LIN {X 0,Y 641.298,Z 835.183,A -85,B 0,C 180,E1 28744.796,E2 28744.796} C_VEL
LIN {X 0,Y 639.476,Z 856.383,A -85,B 0,C 180,E1 28743.716,E2 28743.716} C_VEL
LIN {X 0,Y 637.654,Z 876.672,A -85,B 0,C 180,E1 28742.537,E2 28742.537} C_VEL
LIN {X 0,Y 635.475,Z 900.138,A -85,B 0,C 180,E1 28740.959,E2 28740.959} C_VEL
LIN {X 0,Y 633.786,Z 917.988,A -85,B 0,C 180,E1 28739.591,E2 28739.591} C_VEL
LIN {X 0,Y 632.015,Z 936.849,A -85,B 0,C 180,E1 28737.975,E2 28737.975} C_VEL
LIN {X 0,Y 630.246,Z 955.886,A -85,B 0,C 180,E1 28736.108,E2 28736.108} C_VEL
LIN {X 0,Y 628.902,Z 971.248,A -85,B 0,C 180,E1 28734.417,E2 28734.417} C_VEL
LIN {X 0,Y 627.491,Z 988.385,A -85,B 0,C 180,E1 28732.287,E2 28732.287} C_VEL
LIN {X 0,Y 626.478,Z 1001.923,A -85,B 0,C 180,E1 28730.361,E2 28730.361} C_VEL
LIN {X 0,Y 625.634,Z 1015.034,A -85,B 0,C 180,E1 28728.255,E2 28728.255} C_VEL
LIN {X 0,Y 624.945,Z 1027.385,A -85,B 0,C 180,E1 28725.933,E2 28725.933} C_VEL
LIN {X 0,Y 624.537,Z 1036.289,A -85,B 0,C 180,E1 28723.99,E2 28723.99} C_VEL
LIN {X 0,Y 624.242,Z 1045.129,A -85,B 0,C 180,E1 28721.737,E2 28721.737} C_VEL
LIN {X 0,Y 624.044,Z 1052.386,A -85,B 0,C 180,E1 28719.406,E2 28719.406} C_VEL
LIN {X 0,Y 623.966,Z 1057.241,A -85,B 0,C 180,E1 28717.458,E2 28717.458} C_VEL
LIN {X 0,Y 623.913,Z 1061.124,A -85,B 0,C 180,E1 28715.426,E2 28715.426} C_VEL
LIN {X 0,Y 623.915,Z 1064.167,A -85,B 0,C 180,E1 28712.94,E2 28712.94} C_VEL
LIN {X 0,Y 623.908,Z 1065.282,A -85,B 0,C 180,E1 28710.918,E2 28710.918} C_VEL
LIN {X 0,Y 623.913,Z 1065.26,A -85,B 0,C 180,E1 28708.99,E2 28708.99} C_VEL
LIN {X 0,Y 623.908,Z 1063.894,A -85,B 0,C 180,E1 28706.693,E2 28706.693} C_VEL
LIN {X 0,Y 623.91,Z 1060.804,A -85,B 0,C 180,E1 28704.39,E2 28704.39} C_VEL
LIN {X 0,Y 623.968,Z 1057.034,A -85,B 0,C 180,E1 28702.449,E2 28702.449} C_VEL
LIN {X 0,Y 624.044,Z 1052.131,A -85,B 0,C 180,E1 28700.501,E2 28700.501} C_VEL
LIN {X 0,Y 624.249,Z 1044.691,A -85,B 0,C 180,E1 28698.146,E2 28698.146} C_VEL
LIN {X 0,Y 624.542,Z 1036.159,A -85,B 0,C 180,E1 28695.98,E2 28695.98} C_VEL
LIN {X 0,Y 624.955,Z 1027.192,A -85,B 0,C 180,E1 28694.027,E2 28694.027} C_VEL
LIN {X 0,Y 625.655,Z 1014.638,A -85,B 0,C 180,E1 28691.678,E2 28691.678} C_VEL
LIN {X 0,Y 626.478,Z 1001.926,A -85,B 0,C 180,E1 28689.639,E2 28689.639} C_VEL
LIN {X 0,Y 627.49,Z 988.385,A -85,B 0,C 180,E1 28687.713,E2 28687.713} C_VEL
LIN {X 0,Y 628.903,Z 971.248,A -85,B 0,C 180,E1 28685.583,E2 28685.583} C_VEL
LIN {X 0,Y 630.247,Z 955.885,A -85,B 0,C 180,E1 28683.892,E2 28683.892} C_VEL
LIN {X 0,Y 632.014,Z 936.851,A -85,B 0,C 180,E1 28682.025,E2 28682.025} C_VEL
LIN {X 0,Y 633.784,Z 917.986,A -85,B 0,C 180,E1 28680.409,E2 28680.409} C_VEL
LIN {X 0,Y 635.482,Z 900.053,A -85,B 0,C 180,E1 28679.035,E2 28679.035} C_VEL
LIN {X 0,Y 637.655,Z 876.666,A -85,B 0,C 180,E1 28677.463,E2 28677.463} C_VEL
LIN {X 0,Y 639.476,Z 856.385,A -85,B 0,C 180,E1 28676.284,E2 28676.284} C_VEL
LIN {X 0,Y 641.298,Z 835.19,A -85,B 0,C 180,E1 28675.204,E2 28675.204} C_VEL
LIN {X 0,Y 643.222,Z 810.081,A -85,B 0,C 180,E1 28674.123,E2 28674.123} C_VEL
LIN {X 0,Y 644.618,Z 789.698,A -85,B 0,C 180,E1 28673.387,E2 28673.387} C_VEL
LIN {X 0,Y 645.855,Z 769.341,A -85,B 0,C 180,E1 28672.768,E2 28672.768} C_VEL
LIN {X 0,Y 647.121,Z 744.666,A -85,B 0,C 180,E1 28672.163,E2 28672.163} C_VEL
LIN {X 0,Y 648.017,Z 719.173,A -85,B 0,C 180,E1 28671.716,E2 28671.716} C_VEL
LIN {X 0,Y 651.905,Z 492.19,A -85,B 0,C 180,E1 28668.782,E2 28668.782} C_VEL
LIN {X 0,Y 654.852,Z 321.153,A -85,B 0,C 180,E1 28666.527,E2 28666.527} C_VEL
LIN {X 0,Y 651.999,Z 316.125,A -85,B 0,C 180,E1 28666.214,E2 28666.214} C_VEL
LIN {X 0,Y 636.119,Z 291.599,A -85,B 0,C 180,E1 28664.466,E2 28664.466} C_VEL
LIN {X 0,Y 633.043,Z 286.91,A -85,B 0,C 180,E1 28664.089,E2 28664.089} C_VEL
LIN {X 0,Y 626.285,Z 271.766,A -85,B 0,C 180,E1 28662.11,E2 28662.11} C_VEL
LIN {X 0,Y 624.92,Z 268.282,A -85,B 0,C 180,E1 28661.607,E2 28661.607} C_VEL
LIN {X 0,Y 624.891,Z 268.104,A -85,B 0,C 180,E1 28658.368,E2 28658.368} C_VEL
LIN {X 0,Y 624.891,Z 268.132,A -85,B 0,C 180,E1 28655.622,E2 28655.622} C_VEL
LIN {X 0,Y 624.899,Z 268.127,A -85,B 0,C 180,E1 28652.346,E2 28652.346} C_VEL
LIN {X 0,Y 624.882,Z 268.114,A -85,B 0,C 180,E1 28649.633,E2 28649.633} C_VEL
LIN {X 0,Y 624.93,Z 268.128,A -85,B 0,C 180,E1 28646.513,E2 28646.513} C_VEL
LIN {X 0,Y 624.882,Z 268.129,A -85,B 0,C 180,E1 28643.58,E2 28643.58} C_VEL
LIN {X 0,Y 624.942,Z 268.125,A -85,B 0,C 180,E1 28640.512,E2 28640.512} C_VEL
LIN {X 0,Y 624.881,Z 268.136,A -85,B 0,C 180,E1 28637.603,E2 28637.603} C_VEL
LIN {X 0,Y 624.959,Z 268.135,A -85,B 0,C 180,E1 28634.545,E2 28634.545} C_VEL
LIN {X 0,Y 624.88,Z 268.136,A -85,B 0,C 180,E1 28631.538,E2 28631.538} C_VEL
LIN {X 0,Y 624.955,Z 268.121,A -85,B 0,C 180,E1 28628.464,E2 28628.464} C_VEL
LIN {X 0,Y 624.879,Z 268.136,A -85,B 0,C 180,E1 28625.509,E2 28625.509} C_VEL
LIN {X 0,Y 624.949,Z 268.132,A -85,B 0,C 180,E1 28622.476,E2 28622.476} C_VEL
LIN {X 0,Y 624.879,Z 268.131,A -85,B 0,C 180,E1 28619.45,E2 28619.45} C_VEL
LIN {X 0,Y 624.935,Z 268.132,A -85,B 0,C 180,E1 28616.514,E2 28616.514} C_VEL
LIN {X 0,Y 624.883,Z 268.14,A -85,B 0,C 180,E1 28613.477,E2 28613.477} C_VEL
LIN {X 0,Y 624.901,Z 268.124,A -85,B 0,C 180,E1 28610.7,E2 28610.7} C_VEL
LIN {X 0,Y 624.892,Z 268.125,A -85,B 0,C 180,E1 28607.525,E2 28607.525} C_VEL
LIN {X 0,Y 624.89,Z 268.138,A -85,B 0,C 180,E1 28604.765,E2 28604.765} C_VEL
LIN {X 0,Y 624.902,Z 268.141,A -85,B 0,C 180,E1 28601.529,E2 28601.529} C_VEL
LIN {X 0,Y 624.886,Z 268.126,A -85,B 0,C 180,E1 28598.701,E2 28598.701} C_VEL
LIN {X 0,Y 624.909,Z 268.117,A -85,B 0,C 180,E1 28595.517,E2 28595.517} C_VEL
LIN {X 0,Y 624.881,Z 268.096,A -85,B 0,C 180,E1 28592.631,E2 28592.631} C_VEL
LIN {X 0,Y 624.922,Z 268.133,A -85,B 0,C 180,E1 28589.522,E2 28589.522} C_VEL
LIN {X 0,Y 624.877,Z 268.089,A -85,B 0,C 180,E1 28586.602,E2 28586.602} C_VEL
LIN {X 0,Y 624.924,Z 268.134,A -85,B 0,C 180,E1 28583.437,E2 28583.437} C_VEL
LIN {X 0,Y 624.88,Z 268.143,A -85,B 0,C 180,E1 28580.561,E2 28580.561} C_VEL
LIN {X 0,Y 624.945,Z 268.138,A -85,B 0,C 180,E1 28577.525,E2 28577.525} C_VEL
LIN {X 0,Y 624.9,Z 268.29,A -85,B 0,C 180,E1 28574.603,E2 28574.603} C_VEL
LIN {X 0,Y 626.38,Z 271.89,A -85,B 0,C 180,E1 28574.082,E2 28574.082} C_VEL
LIN {X 0,Y 629.674,Z 279.22,A -85,B 0,C 180,E1 28573.142,E2 28573.142} C_VEL
LIN {X 0,Y 642.492,Z 298.119,A -85,B 0,C 180,E1 28571.691,E2 28571.691} C_VEL
LIN {X 0,Y 645.185,Z 303.131,A -85,B 0,C 180,E1 28571.382,E2 28571.382} C_VEL
LIN {X 0,Y 647.257,Z 309.962,A -85,B 0,C 180,E1 28571.1,E2 28571.1} C_VEL
LIN {X 0,Y 648.579,Z 319.651,A -85,B 0,C 180,E1 28570.84,E2 28570.84} C_VEL
LIN {X 0,Y 648.788,Z 330.896,A -85,B 0,C 180,E1 28570.653,E2 28570.653} C_VEL
LIN {X 0,Y 644.506,Z 559.778,A -85,B 0,C 180,E1 28567.632,E2 28567.632} C_VEL
LIN {X 0,Y 641.698,Z 711.144,A -85,B 0,C 180,E1 28565.655,E2 28565.655} C_VEL
LIN {X 0,Y 640.622,Z 738.163,A -85,B 0,C 180,E1 28565.155,E2 28565.155} C_VEL
LIN {X 0,Y 639.385,Z 760.444,A -85,B 0,C 180,E1 28564.594,E2 28564.594} C_VEL
LIN {X 0,Y 638.102,Z 780.164,A -85,B 0,C 180,E1 28563.988,E2 28563.988} C_VEL
LIN {X 0,Y 636.521,Z 801.864,A -85,B 0,C 180,E1 28563.192,E2 28563.192} C_VEL
LIN {X 0,Y 634.429,Z 827.031,A -85,B 0,C 180,E1 28562.081,E2 28562.081} C_VEL
LIN {X 0,Y 632.62,Z 846.884,A -85,B 0,C 180,E1 28561.056,E2 28561.056} C_VEL
LIN {X 0,Y 630.742,Z 866.537,A -85,B 0,C 180,E1 28559.902,E2 28559.902} C_VEL
LIN {X 0,Y 628.384,Z 890.088,A -85,B 0,C 180,E1 28558.306,E2 28558.306} C_VEL
LIN {X 0,Y 626.553,Z 908.246,A -85,B 0,C 180,E1 28556.899,E2 28556.899} C_VEL
LIN {X 0,Y 624.597,Z 927.793,A -85,B 0,C 180,E1 28555.203,E2 28555.203} C_VEL
LIN {X 0,Y 622.739,Z 946.216,A -85,B 0,C 180,E1 28553.365,E2 28553.365} C_VEL
LIN {X 0,Y 621.354,Z 960.958,A -85,B 0,C 180,E1 28551.723,E2 28551.723} C_VEL
LIN {X 0,Y 619.835,Z 977.944,A -85,B 0,C 180,E1 28549.595,E2 28549.595} C_VEL
LIN {X 0,Y 618.72,Z 991.88,A -85,B 0,C 180,E1 28547.59,E2 28547.59} C_VEL
LIN {X 0,Y 617.803,Z 1004.81,A -85,B 0,C 180,E1 28545.488,E2 28545.488} C_VEL
LIN {X 0,Y 617.047,Z 1017.274,A -85,B 0,C 180,E1 28543.121,E2 28543.121} C_VEL
LIN {X 0,Y 616.593,Z 1026.299,A -85,B 0,C 180,E1 28541.126,E2 28541.126} C_VEL
LIN {X 0,Y 616.273,Z 1035.116,A -85,B 0,C 180,E1 28538.85,E2 28538.85} C_VEL
LIN {X 0,Y 616.05,Z 1042.28,A -85,B 0,C 180,E1 28536.524,E2 28536.524} C_VEL
LIN {X 0,Y 615.972,Z 1047.127,A -85,B 0,C 180,E1 28534.562,E2 28534.562} C_VEL
LIN {X 0,Y 615.911,Z 1051.019,A -85,B 0,C 180,E1 28532.512,E2 28532.512} C_VEL
LIN {X 0,Y 615.928,Z 1054.117,A -85,B 0,C 180,E1 28530,E2 28530} C_VEL
LIN {X 0,Y 615.905,Z 1055.288,A -85,B 0,C 180,E1 28527.86,E2 28527.86} C_VEL
LIN {X 0,Y 615.911,Z 1055.253,A -85,B 0,C 180,E1 28525.904,E2 28525.904} C_VEL
LIN {X 0,Y 615.908,Z 1053.865,A -85,B 0,C 180,E1 28523.568,E2 28523.568} C_VEL
LIN {X 0,Y 615.914,Z 1050.721,A -85,B 0,C 180,E1 28521.222,E2 28521.222} C_VEL
LIN {X 0,Y 615.978,Z 1046.892,A -85,B 0,C 180,E1 28519.241,E2 28519.241} C_VEL
LIN {X 0,Y 616.059,Z 1041.648,A -85,B 0,C 180,E1 28517.153,E2 28517.153} C_VEL
LIN {X 0,Y 616.303,Z 1033.651,A -85,B 0,C 180,E1 28514.666,E2 28514.666} C_VEL
LIN {X 0,Y 616.623,Z 1025.692,A -85,B 0,C 180,E1 28512.641,E2 28512.641} C_VEL
LIN {X 0,Y 617.095,Z 1016.36,A -85,B 0,C 180,E1 28510.6,E2 28510.6} C_VEL
LIN {X 0,Y 617.862,Z 1003.777,A -85,B 0,C 180,E1 28508.248,E2 28508.248} C_VEL
LIN {X 0,Y 618.746,Z 991.569,A -85,B 0,C 180,E1 28506.273,E2 28506.273} C_VEL
LIN {X 0,Y 619.937,Z 976.802,A -85,B 0,C 180,E1 28504.158,E2 28504.158} C_VEL
LIN {X 0,Y 621.359,Z 960.912,A -85,B 0,C 180,E1 28502.182,E2 28502.182} C_VEL
LIN {X 0,Y 622.806,Z 945.515,A -85,B 0,C 180,E1 28500.47,E2 28500.47} C_VEL
LIN {X 0,Y 624.771,Z 925.95,A -85,B 0,C 180,E1 28498.542,E2 28498.542} C_VEL
LIN {X 0,Y 626.593,Z 907.856,A -85,B 0,C 180,E1 28496.979,E2 28496.979} C_VEL
LIN {X 0,Y 628.383,Z 890.122,A -85,B 0,C 180,E1 28495.606,E2 28495.606} C_VEL
LIN {X 0,Y 630.709,Z 866.898,A -85,B 0,C 180,E1 28494.03,E2 28494.03} C_VEL
LIN {X 0,Y 632.612,Z 846.974,A -85,B 0,C 180,E1 28492.859,E2 28492.859} C_VEL
LIN {X 0,Y 634.402,Z 827.3,A -85,B 0,C 180,E1 28491.842,E2 28491.842} C_VEL
LIN {X 0,Y 636.452,Z 802.975,A -85,B 0,C 180,E1 28490.762,E2 28490.762} C_VEL
LIN {X 0,Y 638.079,Z 780.542,A -85,B 0,C 180,E1 28489.935,E2 28489.935} C_VEL
LIN {X 0,Y 639.398,Z 760.213,A -85,B 0,C 180,E1 28489.309,E2 28489.309} C_VEL
LIN {X 0,Y 640.682,Z 737.06,A -85,B 0,C 180,E1 28488.729,E2 28488.729} C_VEL
LIN {X 0,Y 641.708,Z 710.735,A -85,B 0,C 180,E1 28488.249,E2 28488.249} C_VEL
LIN {X 0,Y 645.828,Z 487.761,A -85,B 0,C 180,E1 28485.336,E2 28485.336} C_VEL
LIN {X 0,Y 648.868,Z 320.814,A -85,B 0,C 180,E1 28483.112,E2 28483.112} C_VEL
LIN {X 0,Y 635.425,Z 299.635,A -85,B 0,C 180,E1 28481.58,E2 28481.58} C_VEL
LIN {X 0,Y 624.146,Z 283.107,A -85,B 0,C 180,E1 28480.212,E2 28480.212} C_VEL
LIN {X 0,Y 620.894,Z 278.098,A -85,B 0,C 180,E1 28479.742,E2 28479.742} C_VEL
LIN {X 0,Y 617.061,Z 269.498,A -85,B 0,C 180,E1 28478.456,E2 28478.456} C_VEL
LIN {X 0,Y 616.958,Z 269.106,A -85,B 0,C 180,E1 28477.732,E2 28477.732} C_VEL
LIN {X 0,Y 616.95,Z 269.113,A -85,B 0,C 180,E1 28474.897,E2 28474.897} C_VEL
LIN {X 0,Y 616.965,Z 269.122,A -85,B 0,C 180,E1 28471.675,E2 28471.675} C_VEL
LIN {X 0,Y 616.944,Z 269.127,A -85,B 0,C 180,E1 28468.934,E2 28468.934} C_VEL
LIN {X 0,Y 616.989,Z 269.083,A -85,B 0,C 180,E1 28465.845,E2 28465.845} C_VEL
LIN {X 0,Y 616.943,Z 269.13,A -85,B 0,C 180,E1 28462.891,E2 28462.891} C_VEL
LIN {X 0,Y 616.998,Z 269.081,A -85,B 0,C 180,E1 28459.798,E2 28459.798} C_VEL
LIN {X 0,Y 616.942,Z 269.129,A -85,B 0,C 180,E1 28456.865,E2 28456.865} C_VEL
LIN {X 0,Y 617.007,Z 269.076,A -85,B 0,C 180,E1 28453.782,E2 28453.782} C_VEL
LIN {X 0,Y 616.941,Z 269.127,A -85,B 0,C 180,E1 28450.742,E2 28450.742} C_VEL
LIN {X 0,Y 617.006,Z 269.073,A -85,B 0,C 180,E1 28447.636,E2 28447.636} C_VEL
LIN {X 0,Y 616.942,Z 269.12,A -85,B 0,C 180,E1 28444.63,E2 28444.63} C_VEL
LIN {X 0,Y 617.009,Z 269.094,A -85,B 0,C 180,E1 28441.579,E2 28441.579} C_VEL
LIN {X 0,Y 616.939,Z 269.105,A -85,B 0,C 180,E1 28438.607,E2 28438.607} C_VEL
LIN {X 0,Y 617.012,Z 269.114,A -85,B 0,C 180,E1 28435.539,E2 28435.539} C_VEL
LIN {X 0,Y 616.935,Z 269.08,A -85,B 0,C 180,E1 28432.55,E2 28432.55} C_VEL
LIN {X 0,Y 617.012,Z 269.123,A -85,B 0,C 180,E1 28429.543,E2 28429.543} C_VEL
LIN {X 0,Y 616.937,Z 269.081,A -85,B 0,C 180,E1 28426.503,E2 28426.503} C_VEL
LIN {X 0,Y 617.007,Z 269.117,A -85,B 0,C 180,E1 28423.525,E2 28423.525} C_VEL
LIN {X 0,Y 616.942,Z 269.092,A -85,B 0,C 180,E1 28420.496,E2 28420.496} C_VEL
LIN {X 0,Y 616.997,Z 269.115,A -85,B 0,C 180,E1 28417.514,E2 28417.514} C_VEL
LIN {X 0,Y 616.948,Z 269.121,A -85,B 0,C 180,E1 28414.462,E2 28414.462} C_VEL
LIN {X 0,Y 616.972,Z 269.117,A -85,B 0,C 180,E1 28411.643,E2 28411.643} C_VEL
LIN {X 0,Y 616.947,Z 269.097,A -85,B 0,C 180,E1 28408.433,E2 28408.433} C_VEL
LIN {X 0,Y 616.967,Z 269.104,A -85,B 0,C 180,E1 28405.555,E2 28405.555} C_VEL
LIN {X 0,Y 616.946,Z 269.08,A -85,B 0,C 180,E1 28402.337,E2 28402.337} C_VEL
LIN {X 0,Y 616.96,Z 269.134,A -85,B 0,C 180,E1 28399.589,E2 28399.589} C_VEL
LIN {X 0,Y 617.065,Z 269.581,A -85,B 0,C 180,E1 28399.247,E2 28399.247} C_VEL
LIN {X 0,Y 624.445,Z 286.02,A -85,B 0,C 180,E1 28396.864,E2 28396.864} C_VEL
LIN {X 0,Y 627.63,Z 291.141,A -85,B 0,C 180,E1 28396.4,E2 28396.4} C_VEL
LIN {X 0,Y 637.971,Z 306.703,A -85,B 0,C 180,E1 28395.163,E2 28395.163} C_VEL
LIN {X 0,Y 649.065,Z 324.723,A -85,B 0,C 180,E1 28393.904,E2 28393.904} C_VEL
LIN {X 0,Y 644.542,Z 565.677,A -85,B 0,C 180,E1 28390.726,E2 28390.726} C_VEL
LIN {X 0,Y 641.679,Z 720.881,A -85,B 0,C 180,E1 28388.702,E2 28388.702} C_VEL
LIN {X 0,Y 640.605,Z 747.926,A -85,B 0,C 180,E1 28388.202,E2 28388.202} C_VEL
LIN {X 0,Y 639.373,Z 770.221,A -85,B 0,C 180,E1 28387.643,E2 28387.643} C_VEL
LIN {X 0,Y 638.072,Z 790.382,A -85,B 0,C 180,E1 28387.023,E2 28387.023} C_VEL
LIN {X 0,Y 636.408,Z 813.575,A -85,B 0,C 180,E1 28386.17,E2 28386.17} C_VEL
LIN {X 0,Y 634.404,Z 837.274,A -85,B 0,C 180,E1 28385.114,E2 28385.114} C_VEL
LIN {X 0,Y 632.582,Z 857.28,A -85,B 0,C 180,E1 28384.079,E2 28384.079} C_VEL
LIN {X 0,Y 630.574,Z 878.292,A -85,B 0,C 180,E1 28382.84,E2 28382.84} C_VEL
LIN {X 0,Y 628.39,Z 900.057,A -85,B 0,C 180,E1 28381.354,E2 28381.354} C_VEL
LIN {X 0,Y 626.543,Z 918.332,A -85,B 0,C 180,E1 28379.938,E2 28379.938} C_VEL
LIN {X 0,Y 624.582,Z 937.951,A -85,B 0,C 180,E1 28378.233,E2 28378.233} C_VEL
LIN {X 0,Y 622.736,Z 956.235,A -85,B 0,C 180,E1 28376.408,E2 28376.408} C_VEL
LIN {X 0,Y 621.33,Z 971.246,A -85,B 0,C 180,E1 28374.734,E2 28374.734} C_VEL
LIN {X 0,Y 619.796,Z 988.387,A -85,B 0,C 180,E1 28372.579,E2 28372.579} C_VEL
LIN {X 0,Y 618.717,Z 1001.921,A -85,B 0,C 180,E1 28370.628,E2 28370.628} C_VEL
LIN {X 0,Y 617.784,Z 1015.142,A -85,B 0,C 180,E1 28368.477,E2 28368.477} C_VEL
LIN {X 0,Y 617.05,Z 1027.188,A -85,B 0,C 180,E1 28366.183,E2 28366.183} C_VEL
LIN {X 0,Y 616.596,Z 1036.288,A -85,B 0,C 180,E1 28364.174,E2 28364.174} C_VEL
LIN {X 0,Y 616.269,Z 1045.129,A -85,B 0,C 180,E1 28361.891,E2 28361.891} C_VEL
LIN {X 0,Y 616.05,Z 1052.387,A -85,B 0,C 180,E1 28359.529,E2 28359.529} C_VEL
LIN {X 0,Y 615.972,Z 1057.241,A -85,B 0,C 180,E1 28357.555,E2 28357.555} C_VEL
LIN {X 0,Y 615.912,Z 1061.124,A -85,B 0,C 180,E1 28355.496,E2 28355.496} C_VEL
LIN {X 0,Y 615.915,Z 1064.167,A -85,B 0,C 180,E1 28352.978,E2 28352.978} C_VEL
LIN {X 0,Y 615.908,Z 1065.282,A -85,B 0,C 180,E1 28350.93,E2 28350.93} C_VEL
LIN {X 0,Y 615.913,Z 1065.26,A -85,B 0,C 180,E1 28348.977,E2 28348.977} C_VEL
LIN {X 0,Y 615.908,Z 1063.894,A -85,B 0,C 180,E1 28346.65,E2 28346.65} C_VEL
LIN {X 0,Y 615.912,Z 1060.804,A -85,B 0,C 180,E1 28344.317,E2 28344.317} C_VEL
LIN {X 0,Y 615.977,Z 1057.034,A -85,B 0,C 180,E1 28342.351,E2 28342.351} C_VEL
LIN {X 0,Y 616.052,Z 1052.131,A -85,B 0,C 180,E1 28340.376,E2 28340.376} C_VEL
LIN {X 0,Y 616.275,Z 1044.778,A -85,B 0,C 180,E1 28338.014,E2 28338.014} C_VEL
LIN {X 0,Y 616.596,Z 1036.289,A -85,B 0,C 180,E1 28335.826,E2 28335.826} C_VEL
LIN {X 0,Y 617.05,Z 1027.192,A -85,B 0,C 180,E1 28333.817,E2 28333.817} C_VEL
LIN {X 0,Y 617.79,Z 1015.037,A -85,B 0,C 180,E1 28331.505,E2 28331.505} C_VEL
LIN {X 0,Y 618.717,Z 1001.924,A -85,B 0,C 180,E1 28329.372,E2 28329.372} C_VEL
LIN {X 0,Y 619.796,Z 988.387,A -85,B 0,C 180,E1 28327.421,E2 28327.421} C_VEL
LIN {X 0,Y 621.329,Z 971.246,A -85,B 0,C 180,E1 28325.266,E2 28325.266} C_VEL
LIN {X 0,Y 622.737,Z 956.236,A -85,B 0,C 180,E1 28323.592,E2 28323.592} C_VEL
LIN {X 0,Y 624.635,Z 937.404,A -85,B 0,C 180,E1 28321.717,E2 28321.717} C_VEL
LIN {X 0,Y 626.575,Z 917.983,A -85,B 0,C 180,E1 28320.034,E2 28320.034} C_VEL
LIN {X 0,Y 628.457,Z 899.382,A -85,B 0,C 180,E1 28318.597,E2 28318.597} C_VEL
LIN {X 0,Y 630.816,Z 875.77,A -85,B 0,C 180,E1 28317.006,E2 28317.006} C_VEL
LIN {X 0,Y 632.668,Z 856.381,A -85,B 0,C 180,E1 28315.872,E2 28315.872} C_VEL
LIN {X 0,Y 634.507,Z 836.191,A -85,B 0,C 180,E1 28314.832,E2 28314.832} C_VEL
LIN {X 0,Y 636.556,Z 811.356,A -85,B 0,C 180,E1 28313.744,E2 28313.744} C_VEL
LIN {X 0,Y 638.118,Z 789.647,A -85,B 0,C 180,E1 28312.952,E2 28312.952} C_VEL
LIN {X 0,Y 639.475,Z 768.497,A -85,B 0,C 180,E1 28312.308,E2 28312.308} C_VEL
LIN {X 0,Y 640.841,Z 742.232,A -85,B 0,C 180,E1 28311.675,E2 28311.675} C_VEL
LIN {X 0,Y 641.756,Z 718.325,A -85,B 0,C 180,E1 28311.261,E2 28311.261} C_VEL
LIN {X 0,Y 645.947,Z 488.581,A -85,B 0,C 180,E1 28308.266,E2 28308.266} C_VEL
LIN {X 0,Y 648.992,Z 324.32,A -85,B 0,C 180,E1 28306.083,E2 28306.083} C_VEL
LIN {X 0,Y 634.753,Z 302.038,A -85,B 0,C 180,E1 28304.506,E2 28304.506} C_VEL
LIN {X 0,Y 624.632,Z 286.802,A -85,B 0,C 180,E1 28303.309,E2 28303.309} C_VEL
LIN {X 0,Y 619.867,Z 276.24,A -85,B 0,C 180,E1 28301.899,E2 28301.899} C_VEL
LIN {X 0,Y 617.033,Z 269.27,A -85,B 0,C 180,E1 28300.914,E2 28300.914} C_VEL
LIN {X 0,Y 616.94,Z 269.096,A -85,B 0,C 180,E1 28298.016,E2 28298.016} C_VEL
LIN {X 0,Y 617.008,Z 269.092,A -85,B 0,C 180,E1 28295.007,E2 28295.007} C_VEL
LIN {X 0,Y 616.944,Z 269.129,A -85,B 0,C 180,E1 28292.004,E2 28292.004} C_VEL
LIN {X 0,Y 616.99,Z 269.085,A -85,B 0,C 180,E1 28289.09,E2 28289.09} C_VEL
LIN {X 0,Y 616.946,Z 269.13,A -85,B 0,C 180,E1 28285.95,E2 28285.95} C_VEL
LIN {X 0,Y 616.996,Z 269.116,A -85,B 0,C 180,E1 28282.989,E2 28282.989} C_VEL
LIN {X 0,Y 616.947,Z 269.12,A -85,B 0,C 180,E1 28279.898,E2 28279.898} C_VEL
LIN {X 0,Y 616.985,Z 269.117,A -85,B 0,C 180,E1 28276.96,E2 28276.96} C_VEL
LIN {X 0,Y 616.949,Z 269.125,A -85,B 0,C 180,E1 28273.879,E2 28273.879} C_VEL
LIN {X 0,Y 616.965,Z 269.123,A -85,B 0,C 180,E1 28271.025,E2 28271.025} C_VEL
LIN {X 0,Y 616.952,Z 269.121,A -85,B 0,C 180,E1 28267.824,E2 28267.824} C_VEL
LIN {X 0,Y 616.951,Z 269.123,A -85,B 0,C 180,E1 28265.114,E2 28265.114} C_VEL
LIN {X 0,Y 616.962,Z 269.128,A -85,B 0,C 180,E1 28261.857,E2 28261.857} C_VEL
LIN {X 0,Y 616.946,Z 269.119,A -85,B 0,C 180,E1 28259.071,E2 28259.071} C_VEL
LIN {X 0,Y 616.976,Z 269.113,A -85,B 0,C 180,E1 28255.911,E2 28255.911} C_VEL
LIN {X 0,Y 616.945,Z 269.127,A -85,B 0,C 180,E1 28253.018,E2 28253.018} C_VEL
LIN {X 0,Y 616.991,Z 269.122,A -85,B 0,C 180,E1 28249.92,E2 28249.92} C_VEL
LIN {X 0,Y 616.941,Z 269.112,A -85,B 0,C 180,E1 28246.981,E2 28246.981} C_VEL
LIN {X 0,Y 617.003,Z 269.115,A -85,B 0,C 180,E1 28243.912,E2 28243.912} C_VEL
LIN {X 0,Y 616.941,Z 269.128,A -85,B 0,C 180,E1 28240.988,E2 28240.988} C_VEL
LIN {X 0,Y 617.018,Z 269.116,A -85,B 0,C 180,E1 28237.916,E2 28237.916} C_VEL
LIN {X 0,Y 616.936,Z 269.098,A -85,B 0,C 180,E1 28234.956,E2 28234.956} C_VEL
LIN {X 0,Y 617.017,Z 269.092,A -85,B 0,C 180,E1 28231.863,E2 28231.863} C_VEL
LIN {X 0,Y 616.939,Z 269.119,A -85,B 0,C 180,E1 28228.868,E2 28228.868} C_VEL
LIN {X 0,Y 617.009,Z 269.079,A -85,B 0,C 180,E1 28225.783,E2 28225.783} C_VEL
LIN {X 0,Y 616.939,Z 269.119,A -85,B 0,C 180,E1 28222.805,E2 28222.805} C_VEL
LIN {X 0,Y 617.007,Z 269.116,A -85,B 0,C 180,E1 28219.836,E2 28219.836} C_VEL
LIN {X 0,Y 616.942,Z 269.123,A -85,B 0,C 180,E1 28216.829,E2 28216.829} C_VEL
LIN {X 0,Y 617.018,Z 269.384,A -85,B 0,C 180,E1 28215.269,E2 28215.269} C_VEL
LIN {X 0,Y 618.592,Z 273.122,A -85,B 0,C 180,E1 28214.732,E2 28214.732} C_VEL
LIN {X 0,Y 621.311,Z 279.175,A -85,B 0,C 180,E1 28213.931,E2 28213.931} C_VEL
LIN {X 0,Y 637.509,Z 303.066,A -85,B 0,C 180,E1 28212.053,E2 28212.053} C_VEL
LIN {X 0,Y 648.996,Z 321.131,A -85,B 0,C 180,E1 28210.782,E2 28210.782} C_VEL
LIN {X 0,Y 648.788,Z 330.896,A -85,B 0,C 180,E1 28210.653,E2 28210.653} C_VEL
LIN {X 0,Y 647.889,Z 338.599,A -85,B 0,C 180,E1 28210.613,E2 28210.613} C_VEL
LIN {X 0,Y 642.931,Z 359.221,A -85,B 0,C 180,E1 28210.723,E2 28210.723} C_VEL
LIN {X 0,Y 642.245,Z 365.827,A -85,B 0,C 180,E1 28210.682,E2 28210.682} C_VEL
LIN {X 0,Y 638.152,Z 574.867,A -85,B 0,C 180,E1 28207.905,E2 28207.905} C_VEL
LIN {X 0,Y 635.451,Z 711.435,A -85,B 0,C 180,E1 28206.104,E2 28206.104} C_VEL
LIN {X 0,Y 634.285,Z 738.827,A -85,B 0,C 180,E1 28205.59,E2 28205.59} C_VEL
LIN {X 0,Y 632.996,Z 760.796,A -85,B 0,C 180,E1 28205.032,E2 28205.032} C_VEL
LIN {X 0,Y 631.572,Z 781.469,A -85,B 0,C 180,E1 28204.388,E2 28204.388} C_VEL
LIN {X 0,Y 629.731,Z 805.483,A -85,B 0,C 180,E1 28203.488,E2 28203.488} C_VEL
LIN {X 0,Y 627.681,Z 827.908,A -85,B 0,C 180,E1 28202.468,E2 28202.468} C_VEL
LIN {X 0,Y 625.875,Z 846.574,A -85,B 0,C 180,E1 28201.494,E2 28201.494} C_VEL
LIN {X 0,Y 623.946,Z 865.598,A -85,B 0,C 180,E1 28200.371,E2 28200.371} C_VEL
LIN {X 0,Y 621.481,Z 888.7,A -85,B 0,C 180,E1 28198.807,E2 28198.807} C_VEL
LIN {X 0,Y 619.498,Z 906.982,A -85,B 0,C 180,E1 28197.387,E2 28197.387} C_VEL
LIN {X 0,Y 617.623,Z 924.476,A -85,B 0,C 180,E1 28195.868,E2 28195.868} C_VEL
LIN {X 0,Y 615.439,Z 944.8,A -85,B 0,C 180,E1 28193.862,E2 28193.862} C_VEL
LIN {X 0,Y 613.912,Z 959.665,A -85,B 0,C 180,E1 28192.201,E2 28192.201} C_VEL
LIN {X 0,Y 612.43,Z 975.311,A -85,B 0,C 180,E1 28190.25,E2 28190.25} C_VEL
LIN {X 0,Y 611.048,Z 990.903,A -85,B 0,C 180,E1 28188.015,E2 28188.015} C_VEL
LIN {X 0,Y 610.061,Z 1003.361,A -85,B 0,C 180,E1 28185.983,E2 28185.983} C_VEL
LIN {X 0,Y 609.209,Z 1016.147,A -85,B 0,C 180,E1 28183.574,E2 28183.574} C_VEL
LIN {X 0,Y 608.696,Z 1025.672,A -85,B 0,C 180,E1 28181.465,E2 28181.465} C_VEL
LIN {X 0,Y 608.337,Z 1033.807,A -85,B 0,C 180,E1 28179.365,E2 28179.365} C_VEL
LIN {X 0,Y 608.075,Z 1041.63,A -85,B 0,C 180,E1 28176.894,E2 28176.894} C_VEL
LIN {X 0,Y 607.983,Z 1046.804,A -85,B 0,C 180,E1 28174.811,E2 28174.811} C_VEL
LIN {X 0,Y 607.92,Z 1050.611,A -85,B 0,C 180,E1 28172.828,E2 28172.828} C_VEL
LIN {X 0,Y 607.917,Z 1053.661,A -85,B 0,C 180,E1 28170.565,E2 28170.565} C_VEL
LIN {X 0,Y 607.912,Z 1055.23,A -85,B 0,C 180,E1 28168.115,E2 28168.115} C_VEL
LIN {X 0,Y 607.9,Z 1055.311,A -85,B 0,C 180,E1 28166.133,E2 28166.133} C_VEL
LIN {X 0,Y 607.914,Z 1054.317,A -85,B 0,C 180,E1 28164.147,E2 28164.147} C_VEL
LIN {X 0,Y 607.925,Z 1051.769,A -85,B 0,C 180,E1 28161.773,E2 28161.773} C_VEL
LIN {X 0,Y 607.976,Z 1047.428,A -85,B 0,C 180,E1 28159.386,E2 28159.386} C_VEL
LIN {X 0,Y 608.058,Z 1042.567,A -85,B 0,C 180,E1 28157.367,E2 28157.367} C_VEL
LIN {X 0,Y 608.266,Z 1036.197,A -85,B 0,C 180,E1 28155.239,E2 28155.239} C_VEL
LIN {X 0,Y 608.62,Z 1027.155,A -85,B 0,C 180,E1 28152.799,E2 28152.799} C_VEL
LIN {X 0,Y 609.111,Z 1017.948,A -85,B 0,C 180,E1 28150.717,E2 28150.717} C_VEL
LIN {X 0,Y 609.824,Z 1006.916,A -85,B 0,C 180,E1 28148.553,E2 28148.553} C_VEL
LIN {X 0,Y 610.852,Z 993.222,A -85,B 0,C 180,E1 28146.255,E2 28146.255} C_VEL
LIN {X 0,Y 611.954,Z 980.272,A -85,B 0,C 180,E1 28144.343,E2 28144.343} C_VEL
LIN {X 0,Y 613.525,Z 963.984,A -85,B 0,C 180,E1 28142.218,E2 28142.218} C_VEL
LIN {X 0,Y 615.166,Z 947.407,A -85,B 0,C 180,E1 28140.328,E2 28140.328} C_VEL
LIN {X 0,Y 616.912,Z 930.947,A -85,B 0,C 180,E1 28138.649,E2 28138.649} C_VEL
LIN {X 0,Y 619.193,Z 909.986,A -85,B 0,C 180,E1 28136.771,E2 28136.771} C_VEL
LIN {X 0,Y 621.125,Z 891.967,A -85,B 0,C 180,E1 28135.347,E2 28135.347} C_VEL
LIN {X 0,Y 623.381,Z 871.078,A -85,B 0,C 180,E1 28133.881,E2 28133.881} C_VEL
LIN {X 0,Y 625.638,Z 848.938,A -85,B 0,C 180,E1 28132.547,E2 28132.547} C_VEL
LIN {X 0,Y 627.52,Z 829.522,A -85,B 0,C 180,E1 28131.522,E2 28131.522} C_VEL
LIN {X 0,Y 629.496,Z 807.971,A -85,B 0,C 180,E1 28130.531,E2 28130.531} C_VEL
LIN {X 0,Y 631.459,Z 783.259,A -85,B 0,C 180,E1 28129.583,E2 28129.583} C_VEL
LIN {X 0,Y 632.904,Z 762.267,A -85,B 0,C 180,E1 28128.92,E2 28128.92} C_VEL
LIN {X 0,Y 634.095,Z 742.244,A -85,B 0,C 180,E1 28128.401,E2 28128.401} C_VEL
LIN {X 0,Y 635.245,Z 718.747,A -85,B 0,C 180,E1 28127.922,E2 28127.922} C_VEL
LIN {X 0,Y 636.173,Z 680.837,A -85,B 0,C 180,E1 28127.389,E2 28127.389} C_VEL
LIN {X 0,Y 640.582,Z 449.858,A -85,B 0,C 180,E1 28124.354,E2 28124.354} C_VEL
LIN {X 0,Y 643.083,Z 324.418,A -85,B 0,C 180,E1 28122.664,E2 28122.664} C_VEL
LIN {X 0,Y 630.857,Z 305.063,A -85,B 0,C 180,E1 28121.235,E2 28121.235} C_VEL
LIN {X 0,Y 619.328,Z 287.97,A -85,B 0,C 180,E1 28119.803,E2 28119.803} C_VEL
LIN {X 0,Y 612.906,Z 278.785,A -85,B 0,C 180,E1 28118.939,E2 28118.939} C_VEL
LIN {X 0,Y 610.017,Z 273.02,A -85,B 0,C 180,E1 28118.047,E2 28118.047} C_VEL
LIN {X 0,Y 609.03,Z 270.249,A -85,B 0,C 180,E1 28117.578,E2 28117.578} C_VEL
LIN {X 0,Y 609.03,Z 270.095,A -85,B 0,C 180,E1 28114.662,E2 28114.662} C_VEL
LIN {X 0,Y 609.009,Z 270.107,A -85,B 0,C 180,E1 28111.474,E2 28111.474} C_VEL
LIN {X 0,Y 609.016,Z 270.117,A -85,B 0,C 180,E1 28108.75,E2 28108.75} C_VEL
LIN {X 0,Y 609.009,Z 270.075,A -85,B 0,C 180,E1 28105.445,E2 28105.445} C_VEL
LIN {X 0,Y 609.021,Z 270.12,A -85,B 0,C 180,E1 28102.593,E2 28102.593} C_VEL
LIN {X 0,Y 609.014,Z 270.077,A -85,B 0,C 180,E1 28099.369,E2 28099.369} C_VEL
LIN {X 0,Y 609.02,Z 270.12,A -85,B 0,C 180,E1 28096.501,E2 28096.501} C_VEL
LIN {X 0,Y 609.007,Z 270.072,A -85,B 0,C 180,E1 28093.192,E2 28093.192} C_VEL
LIN {X 0,Y 609.028,Z 270.117,A -85,B 0,C 180,E1 28090.309,E2 28090.309} C_VEL
LIN {X 0,Y 609.005,Z 270.062,A -85,B 0,C 180,E1 28087.073,E2 28087.073} C_VEL
LIN {X 0,Y 609.024,Z 270.11,A -85,B 0,C 180,E1 28084.237,E2 28084.237} C_VEL
LIN {X 0,Y 609.011,Z 270.078,A -85,B 0,C 180,E1 28081.035,E2 28081.035} C_VEL
LIN {X 0,Y 609.016,Z 270.096,A -85,B 0,C 180,E1 28078.212,E2 28078.212} C_VEL
LIN {X 0,Y 609.013,Z 270.102,A -85,B 0,C 180,E1 28074.914,E2 28074.914} C_VEL
LIN {X 0,Y 609.016,Z 270.071,A -85,B 0,C 180,E1 28072.073,E2 28072.073} C_VEL
LIN {X 0,Y 609.015,Z 270.11,A -85,B 0,C 180,E1 28068.829,E2 28068.829} C_VEL
LIN {X 0,Y 609.018,Z 270.064,A -85,B 0,C 180,E1 28065.937,E2 28065.937} C_VEL
LIN {X 0,Y 609.016,Z 270.114,A -85,B 0,C 180,E1 28062.712,E2 28062.712} C_VEL
LIN {X 0,Y 609.021,Z 270.069,A -85,B 0,C 180,E1 28059.832,E2 28059.832} C_VEL
LIN {X 0,Y 609.014,Z 270.118,A -85,B 0,C 180,E1 28056.589,E2 28056.589} C_VEL
LIN {X 0,Y 609.032,Z 270.114,A -85,B 0,C 180,E1 28053.687,E2 28053.687} C_VEL
LIN {X 0,Y 609.016,Z 270.119,A -85,B 0,C 180,E1 28050.477,E2 28050.477} C_VEL
LIN {X 0,Y 609.02,Z 270.064,A -85,B 0,C 180,E1 28047.64,E2 28047.64} C_VEL
LIN {X 0,Y 609.015,Z 270.12,A -85,B 0,C 180,E1 28044.349,E2 28044.349} C_VEL
LIN {X 0,Y 609.035,Z 270.062,A -85,B 0,C 180,E1 28041.396,E2 28041.396} C_VEL
LIN {X 0,Y 609.038,Z 270.349,A -85,B 0,C 180,E1 28040.094,E2 28040.094} C_VEL
LIN {X 0,Y 610.396,Z 273.709,A -85,B 0,C 180,E1 28039.557,E2 28039.557} C_VEL
LIN {X 0,Y 615.01,Z 283.555,A -85,B 0,C 180,E1 28038.071,E2 28038.071} C_VEL
LIN {X 0,Y 616.888,Z 287.227,A -85,B 0,C 180,E1 28037.57,E2 28037.57} C_VEL
LIN {X 0,Y 629.695,Z 306.4,A -85,B 0,C 180,E1 28035.949,E2 28035.949} C_VEL
LIN {X 0,Y 642.735,Z 327.045,A -85,B 0,C 180,E1 28034.418,E2 28034.418} C_VEL
LIN {X 0,Y 643.239,Z 328.506,A -85,B 0,C 180,E1 28034.351,E2 28034.351} C_VEL
LIN {X 0,Y 638.436,Z 567.626,A -85,B 0,C 180,E1 28031.17,E2 28031.17} C_VEL
LIN {X 0,Y 635.429,Z 720.777,A -85,B 0,C 180,E1 28029.155,E2 28029.155} C_VEL
LIN {X 0,Y 634.287,Z 747.83,A -85,B 0,C 180,E1 28028.653,E2 28028.653} C_VEL
LIN {X 0,Y 632.966,Z 770.421,A -85,B 0,C 180,E1 28028.081,E2 28028.081} C_VEL
LIN {X 0,Y 631.554,Z 791.031,A -85,B 0,C 180,E1 28027.442,E2 28027.442} C_VEL
LIN {X 0,Y 629.72,Z 815.201,A -85,B 0,C 180,E1 28026.539,E2 28026.539} C_VEL
LIN {X 0,Y 627.653,Z 838.016,A -85,B 0,C 180,E1 28025.506,E2 28025.506} C_VEL
LIN {X 0,Y 625.893,Z 856.375,A -85,B 0,C 180,E1 28024.55,E2 28024.55} C_VEL
LIN {X 0,Y 624.004,Z 875.042,A -85,B 0,C 180,E1 28023.45,E2 28023.45} C_VEL
LIN {X 0,Y 621.638,Z 897.383,A -85,B 0,C 180,E1 28021.95,E2 28021.95} C_VEL
LIN {X 0,Y 619.518,Z 916.767,A -85,B 0,C 180,E1 28020.45,E2 28020.45} C_VEL
LIN {X 0,Y 617.635,Z 934.359,A -85,B 0,C 180,E1 28018.923,E2 28018.923} C_VEL
LIN {X 0,Y 615.488,Z 954.382,A -85,B 0,C 180,E1 28016.952,E2 28016.952} C_VEL
LIN {X 0,Y 613.921,Z 969.554,A -85,B 0,C 180,E1 28015.259,E2 28015.259} C_VEL
LIN {X 0,Y 612.415,Z 985.485,A -85,B 0,C 180,E1 28013.273,E2 28013.273} C_VEL
LIN {X 0,Y 611.067,Z 1000.649,A -85,B 0,C 180,E1 28011.099,E2 28011.099} C_VEL
LIN {X 0,Y 610.104,Z 1012.737,A -85,B 0,C 180,E1 28009.134,E2 28009.134} C_VEL
LIN {X 0,Y 609.261,Z 1025.335,A -85,B 0,C 180,E1 28006.789,E2 28006.789} C_VEL
LIN {X 0,Y 608.726,Z 1035.088,A -85,B 0,C 180,E1 28004.649,E2 28004.649} C_VEL
LIN {X 0,Y 608.368,Z 1043.013,A -85,B 0,C 180,E1 28002.626,E2 28002.626} C_VEL
LIN {X 0,Y 608.109,Z 1050.856,A -85,B 0,C 180,E1 28000.229,E2 28000.229} C_VEL
LIN {X 0,Y 607.988,Z 1056.621,A -85,B 0,C 180,E1 27997.941,E2 27997.941} C_VEL
LIN {X 0,Y 607.924,Z 1060.486,A -85,B 0,C 180,E1 27995.948,E2 27995.948} C_VEL
LIN {X 0,Y 607.914,Z 1063.356,A -85,B 0,C 180,E1 27993.867,E2 27993.867} C_VEL
LIN {X 0,Y 607.906,Z 1065.191,A -85,B 0,C 180,E1 27991.32,E2 27991.32} C_VEL
LIN {X 0,Y 607.899,Z 1065.327,A -85,B 0,C 180,E1 27989.246,E2 27989.246} C_VEL
LIN {X 0,Y 607.913,Z 1064.37,A -85,B 0,C 180,E1 27987.266,E2 27987.266} C_VEL
LIN {X 0,Y 607.917,Z 1061.994,A -85,B 0,C 180,E1 27984.999,E2 27984.999} C_VEL
LIN {X 0,Y 607.973,Z 1057.654,A -85,B 0,C 180,E1 27982.535,E2 27982.535} C_VEL
LIN {X 0,Y 608.057,Z 1052.895,A -85,B 0,C 180,E1 27980.535,E2 27980.535} C_VEL
LIN {X 0,Y 608.23,Z 1046.969,A -85,B 0,C 180,E1 27978.527,E2 27978.527} C_VEL
LIN {X 0,Y 608.592,Z 1037.907,A -85,B 0,C 180,E1 27976.024,E2 27976.024} C_VEL
LIN {X 0,Y 609.075,Z 1028.567,A -85,B 0,C 180,E1 27973.893,E2 27973.893} C_VEL
LIN {X 0,Y 609.722,Z 1018.24,A -85,B 0,C 180,E1 27971.846,E2 27971.846} C_VEL
LIN {X 0,Y 610.767,Z 1004.262,A -85,B 0,C 180,E1 27969.46,E2 27969.46} C_VEL
LIN {X 0,Y 611.874,Z 991.198,A -85,B 0,C 180,E1 27967.518,E2 27967.518} C_VEL
LIN {X 0,Y 613.381,Z 975.447,A -85,B 0,C 180,E1 27965.438,E2 27965.438} C_VEL
LIN {X 0,Y 615.098,Z 958.086,A -85,B 0,C 180,E1 27963.447,E2 27963.447} C_VEL
LIN {X 0,Y 616.801,Z 941.895,A -85,B 0,C 180,E1 27961.787,E2 27961.787} C_VEL
LIN {X 0,Y 619.146,Z 920.415,A -85,B 0,C 180,E1 27959.851,E2 27959.851} C_VEL
LIN {X 0,Y 621.045,Z 902.718,A -85,B 0,C 180,E1 27958.45,E2 27958.45} C_VEL
LIN {X 0,Y 623.17,Z 882.875,A -85,B 0,C 180,E1 27957.049,E2 27957.049} C_VEL
LIN {X 0,Y 625.534,Z 859.978,A -85,B 0,C 180,E1 27955.65,E2 27955.65} C_VEL
LIN {X 0,Y 627.345,Z 841.19,A -85,B 0,C 180,E1 27954.651,E2 27954.651} C_VEL
LIN {X 0,Y 629.079,Z 821.937,A -85,B 0,C 180,E1 27953.753,E2 27953.753} C_VEL
LIN {X 0,Y 631.127,Z 797.709,A -85,B 0,C 180,E1 27952.786,E2 27952.786} C_VEL
LIN {X 0,Y 632.778,Z 773.544,A -85,B 0,C 180,E1 27952.008,E2 27952.008} C_VEL
LIN {X 0,Y 633.965,Z 753.724,A -85,B 0,C 180,E1 27951.487,E2 27951.487} C_VEL
LIN {X 0,Y 634.965,Z 733.427,A -85,B 0,C 180,E1 27951.06,E2 27951.06} C_VEL
LIN {X 0,Y 635.877,Z 705.307,A -85,B 0,C 180,E1 27950.626,E2 27950.626} C_VEL
LIN {X 0,Y 640.401,Z 466.376,A -85,B 0,C 180,E1 27947.493,E2 27947.493} C_VEL
LIN {X 0,Y 643.083,Z 327.703,A -85,B 0,C 180,E1 27945.63,E2 27945.63} C_VEL
LIN {X 0,Y 627.268,Z 303.03,A -85,B 0,C 180,E1 27943.837,E2 27943.837} C_VEL
LIN {X 0,Y 616.356,Z 286.61,A -85,B 0,C 180,E1 27942.507,E2 27942.507} C_VEL
LIN {X 0,Y 610.233,Z 273.424,A -85,B 0,C 180,E1 27940.656,E2 27940.656} C_VEL
LIN {X 0,Y 609.029,Z 270.281,A -85,B 0,C 180,E1 27940.182,E2 27940.182} C_VEL
LIN {X 0,Y 609.02,Z 270.09,A -85,B 0,C 180,E1 27937.525,E2 27937.525} C_VEL
LIN {X 0,Y 609.012,Z 270.074,A -85,B 0,C 180,E1 27934.274,E2 27934.274} C_VEL
LIN {X 0,Y 609.025,Z 270.118,A -85,B 0,C 180,E1 27931.381,E2 27931.381} C_VEL
LIN {X 0,Y 609.007,Z 270.077,A -85,B 0,C 180,E1 27928.113,E2 27928.113} C_VEL
LIN {X 0,Y 609.032,Z 270.117,A -85,B 0,C 180,E1 27925.23,E2 27925.23} C_VEL
LIN {X 0,Y 609.012,Z 270.118,A -85,B 0,C 180,E1 27921.983,E2 27921.983} C_VEL
LIN {X 0,Y 609.035,Z 270.11,A -85,B 0,C 180,E1 27919.069,E2 27919.069} C_VEL
LIN {X 0,Y 609.011,Z 270.11,A -85,B 0,C 180,E1 27915.914,E2 27915.914} C_VEL
LIN {X 0,Y 609.023,Z 270.108,A -85,B 0,C 180,E1 27913.095,E2 27913.095} C_VEL
LIN {X 0,Y 609.011,Z 270.114,A -85,B 0,C 180,E1 27909.831,E2 27909.831} C_VEL
LIN {X 0,Y 609.023,Z 270.111,A -85,B 0,C 180,E1 27906.978,E2 27906.978} C_VEL
LIN {X 0,Y 609.014,Z 270.106,A -85,B 0,C 180,E1 27903.765,E2 27903.765} C_VEL
LIN {X 0,Y 609.028,Z 270.113,A -85,B 0,C 180,E1 27900.847,E2 27900.847} C_VEL
LIN {X 0,Y 609.012,Z 270.118,A -85,B 0,C 180,E1 27897.648,E2 27897.648} C_VEL
LIN {X 0,Y 609.029,Z 270.103,A -85,B 0,C 180,E1 27894.725,E2 27894.725} C_VEL
LIN {X 0,Y 609.008,Z 270.101,A -85,B 0,C 180,E1 27891.503,E2 27891.503} C_VEL
LIN {X 0,Y 609.03,Z 270.115,A -85,B 0,C 180,E1 27888.638,E2 27888.638} C_VEL
LIN {X 0,Y 609.014,Z 270.119,A -85,B 0,C 180,E1 27885.451,E2 27885.451} C_VEL
LIN {X 0,Y 609.019,Z 270.1,A -85,B 0,C 180,E1 27882.614,E2 27882.614} C_VEL
LIN {X 0,Y 609.01,Z 270.103,A -85,B 0,C 180,E1 27879.329,E2 27879.329} C_VEL
LIN {X 0,Y 609.015,Z 270.116,A -85,B 0,C 180,E1 27876.589,E2 27876.589} C_VEL
LIN {X 0,Y 609.007,Z 270.058,A -85,B 0,C 180,E1 27873.265,E2 27873.265} C_VEL
LIN {X 0,Y 609.017,Z 270.116,A -85,B 0,C 180,E1 27870.476,E2 27870.476} C_VEL
LIN {X 0,Y 609.008,Z 270.061,A -85,B 0,C 180,E1 27867.193,E2 27867.193} C_VEL
LIN {X 0,Y 609.019,Z 270.116,A -85,B 0,C 180,E1 27864.349,E2 27864.349} C_VEL
LIN {X 0,Y 609.011,Z 270.115,A -85,B 0,C 180,E1 27861.037,E2 27861.037} C_VEL
LIN {X 0,Y 609.011,Z 270.105,A -85,B 0,C 180,E1 27858.322,E2 27858.322} C_VEL
LIN {X 0,Y 609.06,Z 270.289,A -85,B 0,C 180,E1 27856.017,E2 27856.017} C_VEL
LIN {X 0,Y 612.965,Z 279.236,A -85,B 0,C 180,E1 27854.749,E2 27854.749} C_VEL
LIN {X 0,Y 629.881,Z 303.984,A -85,B 0,C 180,E1 27852.728,E2 27852.728} C_VEL
LIN {X 0,Y 642.041,Z 322.798,A -85,B 0,C 180,E1 27851.353,E2 27851.353} C_VEL
LIN {X 0,Y 643.135,Z 325,A -85,B 0,C 180,E1 27851.225,E2 27851.225} C_VEL
LIN {X 0,Y 642.245,Z 365.827,A -85,B 0,C 180,E1 27850.682,E2 27850.682} C_VEL
LIN {X 0,Y 641.345,Z 373.532,A -85,B 0,C 180,E1 27850.642,E2 27850.642} C_VEL
LIN {X 0,Y 636.344,Z 394.151,A -85,B 0,C 180,E1 27850.755,E2 27850.755} C_VEL
LIN {X 0,Y 635.691,Z 400.755,A -85,B 0,C 180,E1 27850.71,E2 27850.71} C_VEL
LIN {X 0,Y 631.474,Z 606.849,A -85,B 0,C 180,E1 27847.959,E2 27847.959} C_VEL
LIN {X 0,Y 629.237,Z 711.934,A -85,B 0,C 180,E1 27846.558,E2 27846.558} C_VEL
LIN {X 0,Y 627.973,Z 739.688,A -85,B 0,C 180,E1 27846.03,E2 27846.03} C_VEL
LIN {X 0,Y 626.636,Z 761.253,A -85,B 0,C 180,E1 27845.476,E2 27845.476} C_VEL
LIN {X 0,Y 625.124,Z 782.055,A -85,B 0,C 180,E1 27844.821,E2 27844.821} C_VEL
LIN {X 0,Y 623.122,Z 806.513,A -85,B 0,C 180,E1 27843.891,E2 27843.891} C_VEL
LIN {X 0,Y 620.968,Z 828.827,A -85,B 0,C 180,E1 27842.863,E2 27842.863} C_VEL
LIN {X 0,Y 619.062,Z 847.395,A -85,B 0,C 180,E1 27841.881,E2 27841.881} C_VEL
LIN {X 0,Y 616.851,Z 867.881,A -85,B 0,C 180,E1 27840.65,E2 27840.65} C_VEL
LIN {X 0,Y 614.32,Z 889.925,A -85,B 0,C 180,E1 27839.121,E2 27839.121} C_VEL
LIN {X 0,Y 612.226,Z 908.1,A -85,B 0,C 180,E1 27837.687,E2 27837.687} C_VEL
LIN {X 0,Y 610.019,Z 927.668,A -85,B 0,C 180,E1 27835.953,E2 27835.953} C_VEL
LIN {X 0,Y 607.875,Z 946.108,A -85,B 0,C 180,E1 27834.075,E2 27834.075} C_VEL
LIN {X 0,Y 606.263,Z 960.859,A -85,B 0,C 180,E1 27832.394,E2 27832.394} C_VEL
LIN {X 0,Y 604.541,Z 977.794,A -85,B 0,C 180,E1 27830.223,E2 27830.223} C_VEL
LIN {X 0,Y 603.226,Z 991.802,A -85,B 0,C 180,E1 27828.157,E2 27828.157} C_VEL
LIN {X 0,Y 602.187,Z 1004.173,A -85,B 0,C 180,E1 27826.099,E2 27826.099} C_VEL
LIN {X 0,Y 601.28,Z 1016.804,A -85,B 0,C 180,E1 27823.659,E2 27823.659} C_VEL
LIN {X 0,Y 600.761,Z 1025.845,A -85,B 0,C 180,E1 27821.618,E2 27821.618} C_VEL
LIN {X 0,Y 600.379,Z 1033.957,A -85,B 0,C 180,E1 27819.49,E2 27819.49} C_VEL
LIN {X 0,Y 600.091,Z 1041.739,A -85,B 0,C 180,E1 27816.986,E2 27816.986} C_VEL
LIN {X 0,Y 599.988,Z 1046.892,A -85,B 0,C 180,E1 27814.876,E2 27814.876} C_VEL
LIN {X 0,Y 599.924,Z 1050.679,A -85,B 0,C 180,E1 27812.866,E2 27812.866} C_VEL
LIN {X 0,Y 599.914,Z 1053.82,A -85,B 0,C 180,E1 27810.477,E2 27810.477} C_VEL
LIN {X 0,Y 599.912,Z 1055.239,A -85,B 0,C 180,E1 27808.09,E2 27808.09} C_VEL
LIN {X 0,Y 599.903,Z 1055.301,A -85,B 0,C 180,E1 27806.082,E2 27806.082} C_VEL
LIN {X 0,Y 599.917,Z 1054.219,A -85,B 0,C 180,E1 27803.973,E2 27803.973} C_VEL
LIN {X 0,Y 599.913,Z 1051.386,A -85,B 0,C 180,E1 27801.469,E2 27801.469} C_VEL
LIN {X 0,Y 599.983,Z 1047.339,A -85,B 0,C 180,E1 27799.243,E2 27799.243} C_VEL
LIN {X 0,Y 600.07,Z 1042.456,A -85,B 0,C 180,E1 27797.196,E2 27797.196} C_VEL
LIN {X 0,Y 600.309,Z 1035.756,A -85,B 0,C 180,E1 27794.94,E2 27794.94} C_VEL
LIN {X 0,Y 600.708,Z 1026.752,A -85,B 0,C 180,E1 27792.511,E2 27792.511} C_VEL
LIN {X 0,Y 601.218,Z 1017.822,A -85,B 0,C 180,E1 27790.471,E2 27790.471} C_VEL
LIN {X 0,Y 602.048,Z 1006.155,A -85,B 0,C 180,E1 27788.16,E2 27788.16} C_VEL
LIN {X 0,Y 603.131,Z 992.936,A -85,B 0,C 180,E1 27785.932,E2 27785.932} C_VEL
LIN {X 0,Y 604.308,Z 979.954,A -85,B 0,C 180,E1 27783.994,E2 27783.994} C_VEL
LIN {X 0,Y 606.082,Z 962.735,A -85,B 0,C 180,E1 27781.74,E2 27781.74} C_VEL
LIN {X 0,Y 607.781,Z 946.916,A -85,B 0,C 180,E1 27779.923,E2 27779.923} C_VEL
LIN {X 0,Y 609.795,Z 929.452,A -85,B 0,C 180,E1 27778.131,E2 27778.131} C_VEL
LIN {X 0,Y 612.105,Z 909.246,A -85,B 0,C 180,E1 27776.318,E2 27776.318} C_VEL
LIN {X 0,Y 614.119,Z 891.65,A -85,B 0,C 180,E1 27774.918,E2 27774.918} C_VEL
LIN {X 0,Y 616.644,Z 869.867,A -85,B 0,C 180,E1 27773.384,E2 27773.384} C_VEL
LIN {X 0,Y 618.98,Z 848.189,A -85,B 0,C 180,E1 27772.073,E2 27772.073} C_VEL
LIN {X 0,Y 620.951,Z 829.006,A -85,B 0,C 180,E1 27771.056,E2 27771.056} C_VEL
LIN {X 0,Y 623.146,Z 806.336,A -85,B 0,C 180,E1 27770.012,E2 27770.012} C_VEL
LIN {X 0,Y 625.138,Z 781.866,A -85,B 0,C 180,E1 27769.082,E2 27769.082} C_VEL
LIN {X 0,Y 626.656,Z 760.949,A -85,B 0,C 180,E1 27768.425,E2 27768.425} C_VEL
LIN {X 0,Y 628.066,Z 738.08,A -85,B 0,C 180,E1 27767.842,E2 27767.842} C_VEL
LIN {X 0,Y 629.255,Z 711.272,A -85,B 0,C 180,E1 27767.341,E2 27767.341} C_VEL
LIN {X 0,Y 632.565,Z 553.193,A -85,B 0,C 180,E1 27765.242,E2 27765.242} C_VEL
LIN {X 0,Y 637.426,Z 328.097,A -85,B 0,C 180,E1 27762.214,E2 27762.214} C_VEL
LIN {X 0,Y 624.261,Z 307.165,A -85,B 0,C 180,E1 27760.625,E2 27760.625} C_VEL
LIN {X 0,Y 611.634,Z 288.975,A -85,B 0,C 180,E1 27759.006,E2 27759.006} C_VEL
LIN {X 0,Y 604.398,Z 278.684,A -85,B 0,C 180,E1 27757.983,E2 27757.983} C_VEL
LIN {X 0,Y 602.27,Z 274.424,A -85,B 0,C 180,E1 27757.299,E2 27757.299} C_VEL
LIN {X 0,Y 601.105,Z 271.228,A -85,B 0,C 180,E1 27756.743,E2 27756.743} C_VEL
LIN {X 0,Y 601.072,Z 271.088,A -85,B 0,C 180,E1 27753.524,E2 27753.524} C_VEL
LIN {X 0,Y 601.082,Z 271.081,A -85,B 0,C 180,E1 27750.682,E2 27750.682} C_VEL
LIN {X 0,Y 601.073,Z 271.092,A -85,B 0,C 180,E1 27747.438,E2 27747.438} C_VEL
LIN {X 0,Y 601.09,Z 271.076,A -85,B 0,C 180,E1 27744.507,E2 27744.507} C_VEL
LIN {X 0,Y 601.071,Z 271.079,A -85,B 0,C 180,E1 27741.32,E2 27741.32} C_VEL
LIN {X 0,Y 601.088,Z 271.082,A -85,B 0,C 180,E1 27738.425,E2 27738.425} C_VEL
LIN {X 0,Y 601.072,Z 271.083,A -85,B 0,C 180,E1 27735.238,E2 27735.238} C_VEL
LIN {X 0,Y 601.081,Z 271.073,A -85,B 0,C 180,E1 27732.392,E2 27732.392} C_VEL
LIN {X 0,Y 601.076,Z 271.096,A -85,B 0,C 180,E1 27729.189,E2 27729.189} C_VEL
LIN {X 0,Y 601.069,Z 271.051,A -85,B 0,C 180,E1 27726.399,E2 27726.399} C_VEL
LIN {X 0,Y 601.075,Z 271.103,A -85,B 0,C 180,E1 27723.051,E2 27723.051} C_VEL
LIN {X 0,Y 601.077,Z 271.052,A -85,B 0,C 180,E1 27720.191,E2 27720.191} C_VEL
LIN {X 0,Y 601.076,Z 271.106,A -85,B 0,C 180,E1 27716.949,E2 27716.949} C_VEL
LIN {X 0,Y 601.08,Z 271.062,A -85,B 0,C 180,E1 27714.08,E2 27714.08} C_VEL
LIN {X 0,Y 601.072,Z 271.094,A -85,B 0,C 180,E1 27710.811,E2 27710.811} C_VEL
LIN {X 0,Y 601.089,Z 271.077,A -85,B 0,C 180,E1 27707.901,E2 27707.901} C_VEL
LIN {X 0,Y 601.068,Z 271.076,A -85,B 0,C 180,E1 27704.663,E2 27704.663} C_VEL
LIN {X 0,Y 601.095,Z 271.089,A -85,B 0,C 180,E1 27701.773,E2 27701.773} C_VEL
LIN {X 0,Y 601.068,Z 271.072,A -85,B 0,C 180,E1 27698.532,E2 27698.532} C_VEL
LIN {X 0,Y 601.1,Z 271.097,A -85,B 0,C 180,E1 27695.636,E2 27695.636} C_VEL
LIN {X 0,Y 601.073,Z 271.102,A -85,B 0,C 180,E1 27692.454,E2 27692.454} C_VEL
LIN {X 0,Y 601.093,Z 271.102,A -85,B 0,C 180,E1 27689.623,E2 27689.623} C_VEL
LIN {X 0,Y 601.067,Z 271.056,A -85,B 0,C 180,E1 27686.361,E2 27686.361} C_VEL
LIN {X 0,Y 601.096,Z 271.075,A -85,B 0,C 180,E1 27683.451,E2 27683.451} C_VEL
LIN {X 0,Y 601.172,Z 271.323,A -85,B 0,C 180,E1 27680.923,E2 27680.923} C_VEL
LIN {X 0,Y 602.713,Z 275.063,A -85,B 0,C 180,E1 27680.304,E2 27680.304} C_VEL
LIN {X 0,Y 608.106,Z 286.664,A -85,B 0,C 180,E1 27678.53,E2 27678.53} C_VEL
LIN {X 0,Y 616.754,Z 299.096,A -85,B 0,C 180,E1 27677.37,E2 27677.37} C_VEL
LIN {X 0,Y 628.432,Z 316.821,A -85,B 0,C 180,E1 27675.901,E2 27675.901} C_VEL
LIN {X 0,Y 637.481,Z 331.679,A -85,B 0,C 180,E1 27674.815,E2 27674.815} C_VEL
LIN {X 0,Y 632.379,Z 569.045,A -85,B 0,C 180,E1 27671.629,E2 27671.629} C_VEL
LIN {X 0,Y 629.221,Z 720.674,A -85,B 0,C 180,E1 27669.616,E2 27669.616} C_VEL
LIN {X 0,Y 628.008,Z 747.735,A -85,B 0,C 180,E1 27669.112,E2 27669.112} C_VEL
LIN {X 0,Y 626.6,Z 770.576,A -85,B 0,C 180,E1 27668.531,E2 27668.531} C_VEL
LIN {X 0,Y 625.072,Z 791.681,A -85,B 0,C 180,E1 27667.869,E2 27667.869} C_VEL
LIN {X 0,Y 623.04,Z 816.593,A -85,B 0,C 180,E1 27666.921,E2 27666.921} C_VEL
LIN {X 0,Y 620.92,Z 838.745,A -85,B 0,C 180,E1 27665.904,E2 27665.904} C_VEL
LIN {X 0,Y 619.048,Z 857.205,A -85,B 0,C 180,E1 27664.931,E2 27664.931} C_VEL
LIN {X 0,Y 616.901,Z 877.383,A -85,B 0,C 180,E1 27663.725,E2 27663.725} C_VEL
LIN {X 0,Y 614.307,Z 900.051,A -85,B 0,C 180,E1 27662.157,E2 27662.157} C_VEL
LIN {X 0,Y 612.238,Z 917.981,A -85,B 0,C 180,E1 27660.742,E2 27660.742} C_VEL
LIN {X 0,Y 610.045,Z 937.404,A -85,B 0,C 180,E1 27659.023,E2 27659.023} C_VEL
LIN {X 0,Y 607.862,Z 956.232,A -85,B 0,C 180,E1 27657.106,E2 27657.106} C_VEL
LIN {X 0,Y 606.224,Z 971.242,A -85,B 0,C 180,E1 27655.394,E2 27655.394} C_VEL
LIN {X 0,Y 604.475,Z 988.391,A -85,B 0,C 180,E1 27653.184,E2 27653.184} C_VEL
LIN {X 0,Y 603.216,Z 1001.917,A -85,B 0,C 180,E1 27651.183,E2 27651.183} C_VEL
LIN {X 0,Y 602.164,Z 1014.455,A -85,B 0,C 180,E1 27649.094,E2 27649.094} C_VEL
LIN {X 0,Y 601.276,Z 1026.854,A -85,B 0,C 180,E1 27646.692,E2 27646.692} C_VEL
LIN {X 0,Y 600.755,Z 1035.881,A -85,B 0,C 180,E1 27644.654,E2 27644.654} C_VEL
LIN {X 0,Y 600.368,Z 1044.071,A -85,B 0,C 180,E1 27642.504,E2 27642.504} C_VEL
LIN {X 0,Y 600.085,Z 1051.877,A -85,B 0,C 180,E1 27639.979,E2 27639.979} C_VEL
LIN {X 0,Y 599.992,Z 1056.828,A -85,B 0,C 180,E1 27637.951,E2 27637.951} C_VEL
LIN {X 0,Y 599.931,Z 1060.486,A -85,B 0,C 180,E1 27636.027,E2 27636.027} C_VEL
LIN {X 0,Y 599.915,Z 1063.356,A -85,B 0,C 180,E1 27633.918,E2 27633.918} C_VEL
LIN {X 0,Y 599.9,Z 1065.168,A -85,B 0,C 180,E1 27631.433,E2 27631.433} C_VEL
LIN {X 0,Y 599.896,Z 1065.35,A -85,B 0,C 180,E1 27629.332,E2 27629.332} C_VEL
LIN {X 0,Y 599.912,Z 1064.438,A -85,B 0,C 180,E1 27627.325,E2 27627.325} C_VEL
LIN {X 0,Y 599.906,Z 1062.334,A -85,B 0,C 180,E1 27625.22,E2 27625.22} C_VEL
LIN {X 0,Y 599.974,Z 1058.067,A -85,B 0,C 180,E1 27622.627,E2 27622.627} C_VEL
LIN {X 0,Y 600.064,Z 1053.149,A -85,B 0,C 180,E1 27620.505,E2 27620.505} C_VEL
LIN {X 0,Y 600.234,Z 1047.575,A -85,B 0,C 180,E1 27618.566,E2 27618.566} C_VEL
LIN {X 0,Y 600.571,Z 1039.823,A -85,B 0,C 180,E1 27616.325,E2 27616.325} C_VEL
LIN {X 0,Y 601.122,Z 1029.483,A -85,B 0,C 180,E1 27613.872,E2 27613.872} C_VEL
LIN {X 0,Y 601.765,Z 1019.724,A -85,B 0,C 180,E1 27611.886,E2 27611.886} C_VEL
LIN {X 0,Y 602.8,Z 1006.812,A -85,B 0,C 180,E1 27609.586,E2 27609.586} C_VEL
LIN {X 0,Y 604.067,Z 992.597,A -85,B 0,C 180,E1 27607.417,E2 27607.417} C_VEL
LIN {X 0,Y 605.46,Z 978.549,A -85,B 0,C 180,E1 27605.511,E2 27605.511} C_VEL
LIN {X 0,Y 607.464,Z 959.936,A -85,B 0,C 180,E1 27603.298,E2 27603.298} C_VEL
LIN {X 0,Y 609.17,Z 944.554,A -85,B 0,C 180,E1 27601.682,E2 27601.682} C_VEL
LIN {X 0,Y 611.161,Z 927.418,A -85,B 0,C 180,E1 27600.067,E2 27600.067} C_VEL
LIN {X 0,Y 613.682,Z 905.646,A -85,B 0,C 180,E1 27598.268,E2 27598.268} C_VEL
LIN {X 0,Y 615.794,Z 886.99,A -85,B 0,C 180,E1 27596.914,E2 27596.914} C_VEL
LIN {X 0,Y 618.077,Z 866.416,A -85,B 0,C 180,E1 27595.594,E2 27595.594} C_VEL
LIN {X 0,Y 620.492,Z 843.023,A -85,B 0,C 180,E1 27594.309,E2 27594.309} C_VEL
LIN {X 0,Y 622.41,Z 822.985,A -85,B 0,C 180,E1 27593.359,E2 27593.359} C_VEL
LIN {X 0,Y 624.388,Z 800.758,A -85,B 0,C 180,E1 27592.454,E2 27592.454} C_VEL
LIN {X 0,Y 626.313,Z 775.161,A -85,B 0,C 180,E1 27591.602,E2 27591.602} C_VEL
LIN {X 0,Y 627.625,Z 754.506,A -85,B 0,C 180,E1 27591.049,E2 27591.049} C_VEL
LIN {X 0,Y 628.663,Z 734.682,A -85,B 0,C 180,E1 27590.625,E2 27590.625} C_VEL
LIN {X 0,Y 629.614,Z 709.053,A -85,B 0,C 180,E1 27590.213,E2 27590.213} C_VEL
LIN {X 0,Y 634.454,Z 468.51,A -85,B 0,C 180,E1 27587.032,E2 27587.032} C_VEL
LIN {X 0,Y 637.203,Z 331.218,A -85,B 0,C 180,E1 27585.176,E2 27585.176} C_VEL
LIN {X 0,Y 622.278,Z 307.896,A -85,B 0,C 180,E1 27583.45,E2 27583.45} C_VEL
LIN {X 0,Y 610.144,Z 290.088,A -85,B 0,C 180,E1 27581.977,E2 27581.977} C_VEL
LIN {X 0,Y 607.84,Z 286.45,A -85,B 0,C 180,E1 27581.65,E2 27581.65} C_VEL
LIN {X 0,Y 603.991,Z 278.137,A -85,B 0,C 180,E1 27580.462,E2 27580.462} C_VEL
LIN {X 0,Y 601.132,Z 271.363,A -85,B 0,C 180,E1 27579.45,E2 27579.45} C_VEL
LIN {X 0,Y 601.063,Z 271.07,A -85,B 0,C 180,E1 27577.954,E2 27577.954} C_VEL
LIN {X 0,Y 601.129,Z 271.063,A -85,B 0,C 180,E1 27574.904,E2 27574.904} C_VEL
LIN {X 0,Y 601.065,Z 271.109,A -85,B 0,C 180,E1 27571.826,E2 27571.826} C_VEL
LIN {X 0,Y 601.135,Z 271.052,A -85,B 0,C 180,E1 27568.732,E2 27568.732} C_VEL
LIN {X 0,Y 601.069,Z 271.108,A -85,B 0,C 180,E1 27565.627,E2 27565.627} C_VEL
LIN {X 0,Y 601.121,Z 271.102,A -85,B 0,C 180,E1 27562.494,E2 27562.494} C_VEL
LIN {X 0,Y 601.067,Z 271.1,A -85,B 0,C 180,E1 27559.534,E2 27559.534} C_VEL
LIN {X 0,Y 601.122,Z 271.088,A -85,B 0,C 180,E1 27556.426,E2 27556.426} C_VEL
LIN {X 0,Y 601.064,Z 271.101,A -85,B 0,C 180,E1 27553.468,E2 27553.468} C_VEL
LIN {X 0,Y 601.125,Z 271.105,A -85,B 0,C 180,E1 27550.349,E2 27550.349} C_VEL
LIN {X 0,Y 601.064,Z 271.101,A -85,B 0,C 180,E1 27547.359,E2 27547.359} C_VEL
LIN {X 0,Y 601.126,Z 271.086,A -85,B 0,C 180,E1 27544.293,E2 27544.293} C_VEL
LIN {X 0,Y 601.066,Z 271.103,A -85,B 0,C 180,E1 27541.223,E2 27541.223} C_VEL
LIN {X 0,Y 601.118,Z 271.104,A -85,B 0,C 180,E1 27538.094,E2 27538.094} C_VEL
LIN {X 0,Y 601.068,Z 271.093,A -85,B 0,C 180,E1 27535.037,E2 27535.037} C_VEL
LIN {X 0,Y 601.104,Z 271.088,A -85,B 0,C 180,E1 27531.872,E2 27531.872} C_VEL
LIN {X 0,Y 601.071,Z 271.105,A -85,B 0,C 180,E1 27528.952,E2 27528.952} C_VEL
LIN {X 0,Y 601.099,Z 271.102,A -85,B 0,C 180,E1 27525.748,E2 27525.748} C_VEL
LIN {X 0,Y 601.066,Z 271.089,A -85,B 0,C 180,E1 27522.876,E2 27522.876} C_VEL
LIN {X 0,Y 601.112,Z 271.09,A -85,B 0,C 180,E1 27519.743,E2 27519.743} C_VEL
LIN {X 0,Y 601.064,Z 271.106,A -85,B 0,C 180,E1 27516.884,E2 27516.884} C_VEL
LIN {X 0,Y 601.115,Z 271.038,A -85,B 0,C 180,E1 27513.739,E2 27513.739} C_VEL
LIN {X 0,Y 601.063,Z 271.106,A -85,B 0,C 180,E1 27510.829,E2 27510.829} C_VEL
LIN {X 0,Y 601.128,Z 271.049,A -85,B 0,C 180,E1 27507.841,E2 27507.841} C_VEL
LIN {X 0,Y 601.063,Z 271.095,A -85,B 0,C 180,E1 27504.743,E2 27504.743} C_VEL
LIN {X 0,Y 601.138,Z 271.083,A -85,B 0,C 180,E1 27501.653,E2 27501.653} C_VEL
LIN {X 0,Y 601.061,Z 271.091,A -85,B 0,C 180,E1 27498.612,E2 27498.612} C_VEL
LIN {X 0,Y 601.1,Z 271.361,A -85,B 0,C 180,E1 27496.759,E2 27496.759} C_VEL
LIN {X 0,Y 602.688,Z 275.009,A -85,B 0,C 180,E1 27496.193,E2 27496.193} C_VEL
LIN {X 0,Y 604.915,Z 279.533,A -85,B 0,C 180,E1 27495.559,E2 27495.559} C_VEL
LIN {X 0,Y 624.119,Z 307.583,A -85,B 0,C 180,E1 27493.201,E2 27493.201} C_VEL
LIN {X 0,Y 637.225,Z 327.948,A -85,B 0,C 180,E1 27491.693,E2 27491.693} C_VEL
LIN {X 0,Y 635.691,Z 400.755,A -85,B 0,C 180,E1 27490.71,E2 27490.71} C_VEL
LIN {X 0,Y 634.836,Z 408.455,A -85,B 0,C 180,E1 27490.666,E2 27490.666} C_VEL
LIN {X 0,Y 629.813,Z 429.072,A -85,B 0,C 180,E1 27490.78,E2 27490.78} C_VEL
LIN {X 0,Y 629.126,Z 435.682,A -85,B 0,C 180,E1 27490.738,E2 27490.738} C_VEL
LIN {X 0,Y 624.344,Z 659.208,A -85,B 0,C 180,E1 27487.747,E2 27487.747} C_VEL
LIN {X 0,Y 623.001,Z 714.614,A -85,B 0,C 180,E1 27486.988,E2 27486.988} C_VEL
LIN {X 0,Y 621.677,Z 740.884,A -85,B 0,C 180,E1 27486.47,E2 27486.47} C_VEL
LIN {X 0,Y 620.295,Z 762.027,A -85,B 0,C 180,E1 27485.919,E2 27485.919} C_VEL
LIN {X 0,Y 618.662,Z 783.359,A -85,B 0,C 180,E1 27485.239,E2 27485.239} C_VEL
LIN {X 0,Y 616.429,Z 808.637,A -85,B 0,C 180,E1 27484.253,E2 27484.253} C_VEL
LIN {X 0,Y 614.388,Z 828.767,A -85,B 0,C 180,E1 27483.316,E2 27483.316} C_VEL
LIN {X 0,Y 612.377,Z 847.352,A -85,B 0,C 180,E1 27482.326,E2 27482.326} C_VEL
LIN {X 0,Y 610.13,Z 867.061,A -85,B 0,C 180,E1 27481.134,E2 27481.134} C_VEL
LIN {X 0,Y 607.352,Z 889.864,A -85,B 0,C 180,E1 27479.542,E2 27479.542} C_VEL
LIN {X 0,Y 605.11,Z 908.028,A -85,B 0,C 180,E1 27478.095,E2 27478.095} C_VEL
LIN {X 0,Y 602.768,Z 927.605,A -85,B 0,C 180,E1 27476.342,E2 27476.342} C_VEL
LIN {X 0,Y 600.545,Z 945.6,A -85,B 0,C 180,E1 27474.493,E2 27474.493} C_VEL
LIN {X 0,Y 598.799,Z 960.395,A -85,B 0,C 180,E1 27472.793,E2 27472.793} C_VEL
LIN {X 0,Y 597.049,Z 976.709,A -85,B 0,C 180,E1 27470.693,E2 27470.693} C_VEL
LIN {X 0,Y 595.516,Z 991.451,A -85,B 0,C 180,E1 27468.502,E2 27468.502} C_VEL
LIN {X 0,Y 594.452,Z 1003.311,A -85,B 0,C 180,E1 27466.511,E2 27466.511} C_VEL
LIN {X 0,Y 593.451,Z 1016.093,A -85,B 0,C 180,E1 27464.041,E2 27464.041} C_VEL
LIN {X 0,Y 592.848,Z 1025.618,A -85,B 0,C 180,E1 27461.874,E2 27461.874} C_VEL
LIN {X 0,Y 592.424,Z 1033.787,A -85,B 0,C 180,E1 27459.709,E2 27459.709} C_VEL
LIN {X 0,Y 592.108,Z 1041.848,A -85,B 0,C 180,E1 27457.081,E2 27457.081} C_VEL
LIN {X 0,Y 591.996,Z 1046.775,A -85,B 0,C 180,E1 27455.039,E2 27455.039} C_VEL
LIN {X 0,Y 591.933,Z 1050.588,A -85,B 0,C 180,E1 27453.002,E2 27453.002} C_VEL
LIN {X 0,Y 591.917,Z 1053.645,A -85,B 0,C 180,E1 27450.677,E2 27450.677} C_VEL
LIN {X 0,Y 591.91,Z 1055.226,A -85,B 0,C 180,E1 27448.161,E2 27448.161} C_VEL
LIN {X 0,Y 591.901,Z 1055.314,A -85,B 0,C 180,E1 27446.125,E2 27446.125} C_VEL
LIN {X 0,Y 591.915,Z 1054.327,A -85,B 0,C 180,E1 27444.086,E2 27444.086} C_VEL
LIN {X 0,Y 591.922,Z 1051.789,A -85,B 0,C 180,E1 27441.647,E2 27441.647} C_VEL
LIN {X 0,Y 591.987,Z 1047.458,A -85,B 0,C 180,E1 27439.194,E2 27439.194} C_VEL
LIN {X 0,Y 592.076,Z 1042.859,A -85,B 0,C 180,E1 27437.219,E2 27437.219} C_VEL
LIN {X 0,Y 592.303,Z 1036.857,A -85,B 0,C 180,E1 27435.132,E2 27435.132} C_VEL
LIN {X 0,Y 592.731,Z 1027.618,A -85,B 0,C 180,E1 27432.526,E2 27432.526} C_VEL
LIN {X 0,Y 593.28,Z 1018.549,A -85,B 0,C 180,E1 27430.404,E2 27430.404} C_VEL
LIN {X 0,Y 594.054,Z 1008.196,A -85,B 0,C 180,E1 27428.297,E2 27428.297} C_VEL
LIN {X 0,Y 595.312,Z 993.828,A -85,B 0,C 180,E1 27425.788,E2 27425.788} C_VEL
LIN {X 0,Y 596.54,Z 981.065,A -85,B 0,C 180,E1 27423.843,E2 27423.843} C_VEL
LIN {X 0,Y 598.336,Z 964.943,A -85,B 0,C 180,E1 27421.667,E2 27421.667} C_VEL
LIN {X 0,Y 600.241,Z 948.042,A -85,B 0,C 180,E1 27419.686,E2 27419.686} C_VEL
LIN {X 0,Y 602.174,Z 932.105,A -85,B 0,C 180,E1 27418.016,E2 27418.016} C_VEL
LIN {X 0,Y 604.727,Z 911.441,A -85,B 0,C 180,E1 27416.103,E2 27416.103} C_VEL
LIN {X 0,Y 607.026,Z 892.429,A -85,B 0,C 180,E1 27414.563,E2 27414.563} C_VEL
LIN {X 0,Y 609.395,Z 873.107,A -85,B 0,C 180,E1 27413.172,E2 27413.172} C_VEL
LIN {X 0,Y 612.066,Z 850.229,A -85,B 0,C 180,E1 27411.746,E2 27411.746} C_VEL
LIN {X 0,Y 614.158,Z 830.973,A -85,B 0,C 180,E1 27410.705,E2 27410.705} C_VEL
LIN {X 0,Y 616.049,Z 812.357,A -85,B 0,C 180,E1 27409.822,E2 27409.822} C_VEL
LIN {X 0,Y 618.254,Z 788.985,A -85,B 0,C 180,E1 27408.869,E2 27408.869} C_VEL
LIN {X 0,Y 620.141,Z 764.36,A -85,B 0,C 180,E1 27408.059,E2 27408.059} C_VEL
LIN {X 0,Y 621.496,Z 743.947,A -85,B 0,C 180,E1 27407.514,E2 27407.514} C_VEL
LIN {X 0,Y 622.592,Z 723.822,A -85,B 0,C 180,E1 27407.086,E2 27407.086} C_VEL
LIN {X 0,Y 623.594,Z 695.497,A -85,B 0,C 180,E1 27406.643,E2 27406.643} C_VEL
LIN {X 0,Y 628.719,Z 458.928,A -85,B 0,C 180,E1 27403.481,E2 27403.481} C_VEL
LIN {X 0,Y 631.569,Z 331.442,A -85,B 0,C 180,E1 27401.728,E2 27401.728} C_VEL
LIN {X 0,Y 619.331,Z 311.983,A -85,B 0,C 180,E1 27400.21,E2 27400.21} C_VEL
LIN {X 0,Y 607.776,Z 295.166,A -85,B 0,C 180,E1 27398.694,E2 27398.694} C_VEL
LIN {X 0,Y 599.826,Z 284.19,A -85,B 0,C 180,E1 27397.598,E2 27397.598} C_VEL
LIN {X 0,Y 595.933,Z 278.767,A -85,B 0,C 180,E1 27396.998,E2 27396.998} C_VEL
LIN {X 0,Y 594.315,Z 275.298,A -85,B 0,C 180,E1 27396.434,E2 27396.434} C_VEL
LIN {X 0,Y 593.183,Z 272.237,A -85,B 0,C 180,E1 27395.884,E2 27395.884} C_VEL
LIN {X 0,Y 593.128,Z 272.087,A -85,B 0,C 180,E1 27392.991,E2 27392.991} C_VEL
LIN {X 0,Y 593.167,Z 272.07,A -85,B 0,C 180,E1 27389.82,E2 27389.82} C_VEL
LIN {X 0,Y 593.126,Z 272.062,A -85,B 0,C 180,E1 27386.902,E2 27386.902} C_VEL
LIN {X 0,Y 593.159,Z 272.086,A -85,B 0,C 180,E1 27383.653,E2 27383.653} C_VEL
LIN {X 0,Y 593.123,Z 272.054,A -85,B 0,C 180,E1 27380.837,E2 27380.837} C_VEL
LIN {X 0,Y 593.171,Z 272.086,A -85,B 0,C 180,E1 27377.663,E2 27377.663} C_VEL
LIN {X 0,Y 593.123,Z 272.056,A -85,B 0,C 180,E1 27374.747,E2 27374.747} C_VEL
LIN {X 0,Y 593.173,Z 272.075,A -85,B 0,C 180,E1 27371.572,E2 27371.572} C_VEL
LIN {X 0,Y 593.124,Z 272.066,A -85,B 0,C 180,E1 27368.629,E2 27368.629} C_VEL
LIN {X 0,Y 593.174,Z 272.051,A -85,B 0,C 180,E1 27365.514,E2 27365.514} C_VEL
LIN {X 0,Y 593.128,Z 272.09,A -85,B 0,C 180,E1 27362.512,E2 27362.512} C_VEL
LIN {X 0,Y 593.163,Z 272.04,A -85,B 0,C 180,E1 27359.324,E2 27359.324} C_VEL
LIN {X 0,Y 593.133,Z 272.097,A -85,B 0,C 180,E1 27356.327,E2 27356.327} C_VEL
LIN {X 0,Y 593.141,Z 272.034,A -85,B 0,C 180,E1 27353.029,E2 27353.029} C_VEL
LIN {X 0,Y 593.139,Z 272.088,A -85,B 0,C 180,E1 27350.099,E2 27350.099} C_VEL
LIN {X 0,Y 593.129,Z 272.041,A -85,B 0,C 180,E1 27346.746,E2 27346.746} C_VEL
LIN {X 0,Y 593.152,Z 272.08,A -85,B 0,C 180,E1 27343.85,E2 27343.85} C_VEL
LIN {X 0,Y 593.13,Z 272.052,A -85,B 0,C 180,E1 27340.604,E2 27340.604} C_VEL
LIN {X 0,Y 593.167,Z 272.08,A -85,B 0,C 180,E1 27337.606,E2 27337.606} C_VEL
LIN {X 0,Y 593.129,Z 272.086,A -85,B 0,C 180,E1 27334.408,E2 27334.408} C_VEL
LIN {X 0,Y 593.183,Z 272.078,A -85,B 0,C 180,E1 27331.398,E2 27331.398} C_VEL
LIN {X 0,Y 593.123,Z 272.05,A -85,B 0,C 180,E1 27328.266,E2 27328.266} C_VEL
LIN {X 0,Y 593.189,Z 272.07,A -85,B 0,C 180,E1 27325.174,E2 27325.174} C_VEL
LIN {X 0,Y 593.126,Z 272.064,A -85,B 0,C 180,E1 27322.025,E2 27322.025} C_VEL
LIN {X 0,Y 593.231,Z 272.657,A -85,B 0,C 180,E1 27321.732,E2 27321.732} C_VEL
LIN {X 0,Y 594.779,Z 275.934,A -85,B 0,C 180,E1 27321.167,E2 27321.167} C_VEL
LIN {X 0,Y 599.9,Z 286.735,A -85,B 0,C 180,E1 27319.455,E2 27319.455} C_VEL
LIN {X 0,Y 612.368,Z 304.52,A -85,B 0,C 180,E1 27317.738,E2 27317.738} C_VEL
LIN {X 0,Y 624.753,Z 323.545,A -85,B 0,C 180,E1 27316.148,E2 27316.148} C_VEL
LIN {X 0,Y 631.769,Z 335.38,A -85,B 0,C 180,E1 27315.283,E2 27315.283} C_VEL
LIN {X 0,Y 626.348,Z 571.141,A -85,B 0,C 180,E1 27312.088,E2 27312.088} C_VEL
LIN {X 0,Y 623.051,Z 720.676,A -85,B 0,C 180,E1 27310.086,E2 27310.086} C_VEL
LIN {X 0,Y 621.76,Z 747.836,A -85,B 0,C 180,E1 27309.576,E2 27309.576} C_VEL
LIN {X 0,Y 620.274,Z 770.704,A -85,B 0,C 180,E1 27308.99,E2 27308.99} C_VEL
LIN {X 0,Y 618.677,Z 791.589,A -85,B 0,C 180,E1 27308.331,E2 27308.331} C_VEL
LIN {X 0,Y 616.532,Z 816.555,A -85,B 0,C 180,E1 27307.375,E2 27307.375} C_VEL
LIN {X 0,Y 614.374,Z 837.981,A -85,B 0,C 180,E1 27306.386,E2 27306.386} C_VEL
LIN {X 0,Y 612.326,Z 857.116,A -85,B 0,C 180,E1 27305.371,E2 27305.371} C_VEL
LIN {X 0,Y 610.012,Z 877.702,A -85,B 0,C 180,E1 27304.13,E2 27304.13} C_VEL
LIN {X 0,Y 607.261,Z 900.494,A -85,B 0,C 180,E1 27302.537,E2 27302.537} C_VEL
LIN {X 0,Y 605.101,Z 918.11,A -85,B 0,C 180,E1 27301.133,E2 27301.133} C_VEL
LIN {X 0,Y 602.727,Z 937.952,A -85,B 0,C 180,E1 27299.355,E2 27299.355} C_VEL
LIN {X 0,Y 600.468,Z 956.23,A -85,B 0,C 180,E1 27297.468,E2 27297.468} C_VEL
LIN {X 0,Y 598.705,Z 971.24,A -85,B 0,C 180,E1 27295.736,E2 27295.736} C_VEL
LIN {X 0,Y 596.848,Z 988.391,A -85,B 0,C 180,E1 27293.498,E2 27293.498} C_VEL
LIN {X 0,Y 595.474,Z 1001.915,A -85,B 0,C 180,E1 27291.472,E2 27291.472} C_VEL
LIN {X 0,Y 594.355,Z 1014.453,A -85,B 0,C 180,E1 27289.355,E2 27289.355} C_VEL
LIN {X 0,Y 593.402,Z 1026.725,A -85,B 0,C 180,E1 27286.948,E2 27286.948} C_VEL
LIN {X 0,Y 592.831,Z 1035.88,A -85,B 0,C 180,E1 27284.855,E2 27284.855} C_VEL
LIN {X 0,Y 592.41,Z 1044.071,A -85,B 0,C 180,E1 27282.675,E2 27282.675} C_VEL
LIN {X 0,Y 592.104,Z 1051.932,A -85,B 0,C 180,E1 27280.094,E2 27280.094} C_VEL
LIN {X 0,Y 591.993,Z 1056.828,A -85,B 0,C 180,E1 27278.059,E2 27278.059} C_VEL
LIN {X 0,Y 591.938,Z 1060.486,A -85,B 0,C 180,E1 27276.109,E2 27276.109} C_VEL
LIN {X 0,Y 591.914,Z 1063.469,A -85,B 0,C 180,E1 27273.874,E2 27273.874} C_VEL
LIN {X 0,Y 591.904,Z 1065.191,A -85,B 0,C 180,E1 27271.355,E2 27271.355} C_VEL
LIN {X 0,Y 591.9,Z 1065.327,A -85,B 0,C 180,E1 27269.226,E2 27269.226} C_VEL
LIN {X 0,Y 591.913,Z 1064.369,A -85,B 0,C 180,E1 27267.192,E2 27267.192} C_VEL
LIN {X 0,Y 591.921,Z 1061.993,A -85,B 0,C 180,E1 27264.864,E2 27264.864} C_VEL
LIN {X 0,Y 591.986,Z 1057.654,A -85,B 0,C 180,E1 27262.332,E2 27262.332} C_VEL
LIN {X 0,Y 592.075,Z 1052.895,A -85,B 0,C 180,E1 27260.277,E2 27260.277} C_VEL
LIN {X 0,Y 592.296,Z 1046.969,A -85,B 0,C 180,E1 27258.214,E2 27258.214} C_VEL
LIN {X 0,Y 592.717,Z 1037.905,A -85,B 0,C 180,E1 27255.642,E2 27255.642} C_VEL
LIN {X 0,Y 593.279,Z 1028.564,A -85,B 0,C 180,E1 27253.452,E2 27253.452} C_VEL
LIN {X 0,Y 594.049,Z 1018.239,A -85,B 0,C 180,E1 27251.349,E2 27251.349} C_VEL
LIN {X 0,Y 595.253,Z 1004.459,A -85,B 0,C 180,E1 27248.932,E2 27248.932} C_VEL
LIN {X 0,Y 596.484,Z 991.626,A -85,B 0,C 180,E1 27246.97,E2 27246.97} C_VEL
LIN {X 0,Y 598.102,Z 976.961,A -85,B 0,C 180,E1 27244.973,E2 27244.973} C_VEL
LIN {X 0,Y 600.131,Z 959.004,A -85,B 0,C 180,E1 27242.837,E2 27242.837} C_VEL
LIN {X 0,Y 601.988,Z 943.54,A -85,B 0,C 180,E1 27241.205,E2 27241.205} C_VEL
LIN {X 0,Y 604.435,Z 924.057,A -85,B 0,C 180,E1 27239.369,E2 27239.369} C_VEL
LIN {X 0,Y 606.827,Z 904.04,A -85,B 0,C 180,E1 27237.733,E2 27237.733} C_VEL
LIN {X 0,Y 609.013,Z 885.743,A -85,B 0,C 180,E1 27236.407,E2 27236.407} C_VEL
LIN {X 0,Y 611.651,Z 863.443,A -85,B 0,C 180,E1 27234.985,E2 27234.985} C_VEL
LIN {X 0,Y 613.955,Z 842.027,A -85,B 0,C 180,E1 27233.817,E2 27233.817} C_VEL
LIN {X 0,Y 615.887,Z 822.9,A -85,B 0,C 180,E1 27232.906,E2 27232.906} C_VEL
LIN {X 0,Y 617.893,Z 801.438,A -85,B 0,C 180,E1 27232.024,E2 27232.024} C_VEL
LIN {X 0,Y 619.951,Z 775.681,A -85,B 0,C 180,E1 27231.155,E2 27231.155} C_VEL
LIN {X 0,Y 621.365,Z 754.57,A -85,B 0,C 180,E1 27230.586,E2 27230.586} C_VEL
LIN {X 0,Y 622.443,Z 735.06,A -85,B 0,C 180,E1 27230.165,E2 27230.165} C_VEL
LIN {X 0,Y 623.395,Z 710.932,A -85,B 0,C 180,E1 27229.77,E2 27229.77} C_VEL
LIN {X 0,Y 628.514,Z 471.041,A -85,B 0,C 180,E1 27226.571,E2 27226.571} C_VEL
LIN {X 0,Y 631.444,Z 334.838,A -85,B 0,C 180,E1 27224.722,E2 27224.722} C_VEL
LIN {X 0,Y 615.55,Z 310.086,A -85,B 0,C 180,E1 27222.845,E2 27222.845} C_VEL
LIN {X 0,Y 603.569,Z 292.417,A -85,B 0,C 180,E1 27221.344,E2 27221.344} C_VEL
LIN {X 0,Y 599.472,Z 286.339,A -85,B 0,C 180,E1 27220.778,E2 27220.778} C_VEL
LIN {X 0,Y 594.307,Z 275.24,A -85,B 0,C 180,E1 27219.118,E2 27219.118} C_VEL
LIN {X 0,Y 593.191,Z 272.263,A -85,B 0,C 180,E1 27218.633,E2 27218.633} C_VEL
LIN {X 0,Y 593.134,Z 272.078,A -85,B 0,C 180,E1 27215.655,E2 27215.655} C_VEL
LIN {X 0,Y 593.146,Z 272.074,A -85,B 0,C 180,E1 27212.376,E2 27212.376} C_VEL
LIN {X 0,Y 593.13,Z 272.056,A -85,B 0,C 180,E1 27209.558,E2 27209.558} C_VEL
LIN {X 0,Y 593.148,Z 272.09,A -85,B 0,C 180,E1 27206.259,E2 27206.259} C_VEL
LIN {X 0,Y 593.141,Z 272.083,A -85,B 0,C 180,E1 27203.338,E2 27203.338} C_VEL
LIN {X 0,Y 593.136,Z 272.083,A -85,B 0,C 180,E1 27200.012,E2 27200.012} C_VEL
LIN {X 0,Y 593.156,Z 272.083,A -85,B 0,C 180,E1 27197.057,E2 27197.057} C_VEL
LIN {X 0,Y 593.131,Z 272.091,A -85,B 0,C 180,E1 27193.831,E2 27193.831} C_VEL
LIN {X 0,Y 593.164,Z 272.09,A -85,B 0,C 180,E1 27190.883,E2 27190.883} C_VEL
LIN {X 0,Y 593.127,Z 272.087,A -85,B 0,C 180,E1 27187.653,E2 27187.653} C_VEL
LIN {X 0,Y 593.168,Z 272.08,A -85,B 0,C 180,E1 27184.738,E2 27184.738} C_VEL
LIN {X 0,Y 593.128,Z 272.093,A -85,B 0,C 180,E1 27181.546,E2 27181.546} C_VEL
LIN {X 0,Y 593.167,Z 272.084,A -85,B 0,C 180,E1 27178.648,E2 27178.648} C_VEL
LIN {X 0,Y 593.126,Z 272.079,A -85,B 0,C 180,E1 27175.456,E2 27175.456} C_VEL
LIN {X 0,Y 593.181,Z 272.086,A -85,B 0,C 180,E1 27172.445,E2 27172.445} C_VEL
LIN {X 0,Y 593.127,Z 272.096,A -85,B 0,C 180,E1 27169.313,E2 27169.313} C_VEL
LIN {X 0,Y 593.189,Z 272.075,A -85,B 0,C 180,E1 27166.251,E2 27166.251} C_VEL
LIN {X 0,Y 593.124,Z 272.077,A -85,B 0,C 180,E1 27163.144,E2 27163.144} C_VEL
LIN {X 0,Y 593.193,Z 272.082,A -85,B 0,C 180,E1 27160.093,E2 27160.093} C_VEL
LIN {X 0,Y 593.125,Z 272.095,A -85,B 0,C 180,E1 27156.991,E2 27156.991} C_VEL
LIN {X 0,Y 593.186,Z 272.023,A -85,B 0,C 180,E1 27153.899,E2 27153.899} C_VEL
LIN {X 0,Y 593.125,Z 272.095,A -85,B 0,C 180,E1 27150.837,E2 27150.837} C_VEL
LIN {X 0,Y 593.187,Z 272.034,A -85,B 0,C 180,E1 27147.798,E2 27147.798} C_VEL
LIN {X 0,Y 593.126,Z 272.084,A -85,B 0,C 180,E1 27144.674,E2 27144.674} C_VEL
LIN {X 0,Y 593.182,Z 272.074,A -85,B 0,C 180,E1 27141.537,E2 27141.537} C_VEL
LIN {X 0,Y 593.123,Z 272.079,A -85,B 0,C 180,E1 27138.606,E2 27138.606} C_VEL
LIN {X 0,Y 593.24,Z 272.443,A -85,B 0,C 180,E1 27137.524,E2 27137.524} C_VEL
LIN {X 0,Y 594.768,Z 276.044,A -85,B 0,C 180,E1 27136.957,E2 27136.957} C_VEL
LIN {X 0,Y 596.477,Z 279.716,A -85,B 0,C 180,E1 27136.451,E2 27136.451} C_VEL
LIN {X 0,Y 601.953,Z 287.501,A -85,B 0,C 180,E1 27135.727,E2 27135.727} C_VEL
LIN {X 0,Y 613.315,Z 303.761,A -85,B 0,C 180,E1 27134.299,E2 27134.299} C_VEL
LIN {X 0,Y 629.769,Z 328.807,A -85,B 0,C 180,E1 27132.347,E2 27132.347} C_VEL
LIN {X 0,Y 631.486,Z 332.011,A -85,B 0,C 180,E1 27132.141,E2 27132.141} C_VEL
LIN {X 0,Y 629.126,Z 435.682,A -85,B 0,C 180,E1 27130.738,E2 27130.738} C_VEL
LIN {X 0,Y 628.246,Z 443.383,A -85,B 0,C 180,E1 27130.695,E2 27130.695} C_VEL
LIN {X 0,Y 623.239,Z 464.001,A -85,B 0,C 180,E1 27130.81,E2 27130.81} C_VEL
LIN {X 0,Y 622.547,Z 470.61,A -85,B 0,C 180,E1 27130.767,E2 27130.767} C_VEL
LIN {X 0,Y 617.238,Z 704.354,A -85,B 0,C 180,E1 27127.623,E2 27127.623} C_VEL
LIN {X 0,Y 616.287,Z 726.871,A -85,B 0,C 180,E1 27127.244,E2 27127.244} C_VEL
LIN {X 0,Y 615.124,Z 746.892,A -85,B 0,C 180,E1 27126.802,E2 27126.802} C_VEL
LIN {X 0,Y 613.434,Z 770.92,A -85,B 0,C 180,E1 27126.132,E2 27126.132} C_VEL
LIN {X 0,Y 611.264,Z 795.188,A -85,B 0,C 180,E1 27125.27,E2 27125.27} C_VEL
LIN {X 0,Y 609.291,Z 815.172,A -85,B 0,C 180,E1 27124.426,E2 27124.426} C_VEL
LIN {X 0,Y 606.956,Z 836.924,A -85,B 0,C 180,E1 27123.36,E2 27123.36} C_VEL
LIN {X 0,Y 604.194,Z 859.917,A -85,B 0,C 180,E1 27122.032,E2 27122.032} C_VEL
LIN {X 0,Y 601.833,Z 878.82,A -85,B 0,C 180,E1 27120.778,E2 27120.778} C_VEL
LIN {X 0,Y 599.218,Z 899.506,A -85,B 0,C 180,E1 27119.225,E2 27119.225} C_VEL
LIN {X 0,Y 596.561,Z 919.39,A -85,B 0,C 180,E1 27117.501,E2 27117.501} C_VEL
LIN {X 0,Y 594.452,Z 935.533,A -85,B 0,C 180,E1 27115.933,E2 27115.933} C_VEL
LIN {X 0,Y 592.247,Z 953.264,A -85,B 0,C 180,E1 27114.009,E2 27114.009} C_VEL
LIN {X 0,Y 590.146,Z 970.254,A -85,B 0,C 180,E1 27111.885,E2 27111.885} C_VEL
LIN {X 0,Y 588.6,Z 983.919,A -85,B 0,C 180,E1 27109.965,E2 27109.965} C_VEL
LIN {X 0,Y 587.056,Z 999.017,A -85,B 0,C 180,E1 27107.546,E2 27107.546} C_VEL
LIN {X 0,Y 586.024,Z 1010.51,A -85,B 0,C 180,E1 27105.415,E2 27105.415} C_VEL
LIN {X 0,Y 585.219,Z 1021.273,A -85,B 0,C 180,E1 27103.135,E2 27103.135} C_VEL
LIN {X 0,Y 584.616,Z 1031.112,A -85,B 0,C 180,E1 27100.644,E2 27100.644} C_VEL
LIN {X 0,Y 584.285,Z 1038.007,A -85,B 0,C 180,E1 27098.562,E2 27098.562} C_VEL
LIN {X 0,Y 584.075,Z 1043.977,A -85,B 0,C 180,E1 27096.389,E2 27096.389} C_VEL
LIN {X 0,Y 583.954,Z 1049.542,A -85,B 0,C 180,E1 27093.731,E2 27093.731} C_VEL
LIN {X 0,Y 583.901,Z 1052.676,A -85,B 0,C 180,E1 27091.57,E2 27091.57} C_VEL
LIN {X 0,Y 583.912,Z 1054.571,A -85,B 0,C 180,E1 27089.509,E2 27089.509} C_VEL
LIN {X 0,Y 583.897,Z 1055.439,A -85,B 0,C 180,E1 27087.252,E2 27087.252} C_VEL
LIN {X 0,Y 583.905,Z 1054.775,A -85,B 0,C 180,E1 27084.694,E2 27084.694} C_VEL
LIN {X 0,Y 583.905,Z 1053.001,A -85,B 0,C 180,E1 27082.621,E2 27082.621} C_VEL
LIN {X 0,Y 583.948,Z 1050.125,A -85,B 0,C 180,E1 27080.539,E2 27080.539} C_VEL
LIN {X 0,Y 584.015,Z 1045.877,A -85,B 0,C 180,E1 27078.329,E2 27078.329} C_VEL
LIN {X 0,Y 584.227,Z 1039.176,A -85,B 0,C 180,E1 27075.732,E2 27075.732} C_VEL
LIN {X 0,Y 584.547,Z 1032.313,A -85,B 0,C 180,E1 27073.606,E2 27073.606} C_VEL
LIN {X 0,Y 585.007,Z 1024.15,A -85,B 0,C 180,E1 27071.464,E2 27071.464} C_VEL
LIN {X 0,Y 585.86,Z 1012.522,A -85,B 0,C 180,E1 27068.893,E2 27068.893} C_VEL
LIN {X 0,Y 586.817,Z 1001.577,A -85,B 0,C 180,E1 27066.821,E2 27066.821} C_VEL
LIN {X 0,Y 588.054,Z 989.124,A -85,B 0,C 180,E1 27064.736,E2 27064.736} C_VEL
LIN {X 0,Y 589.786,Z 973.292,A -85,B 0,C 180,E1 27062.43,E2 27062.43} C_VEL
LIN {X 0,Y 591.453,Z 959.375,A -85,B 0,C 180,E1 27060.642,E2 27060.642} C_VEL
LIN {X 0,Y 593.513,Z 943.13,A -85,B 0,C 180,E1 27058.772,E2 27058.772} C_VEL
LIN {X 0,Y 596.03,Z 923.326,A -85,B 0,C 180,E1 27056.774,E2 27056.774} C_VEL
LIN {X 0,Y 598.273,Z 906.321,A -85,B 0,C 180,E1 27055.256,E2 27055.256} C_VEL
LIN {X 0,Y 601.002,Z 885.897,A -85,B 0,C 180,E1 27053.633,E2 27053.633} C_VEL
LIN {X 0,Y 603.694,Z 864.148,A -85,B 0,C 180,E1 27052.146,E2 27052.146} C_VEL
LIN {X 0,Y 605.986,Z 845.092,A -85,B 0,C 180,E1 27051.002,E2 27051.002} C_VEL
LIN {X 0,Y 608.612,Z 821.856,A -85,B 0,C 180,E1 27049.785,E2 27049.785} C_VEL
LIN {X 0,Y 610.948,Z 798.387,A -85,B 0,C 180,E1 27048.765,E2 27048.765} C_VEL
LIN {X 0,Y 612.775,Z 777.871,A -85,B 0,C 180,E1 27048.009,E2 27048.009} C_VEL
LIN {X 0,Y 614.785,Z 752.494,A -85,B 0,C 180,E1 27047.245,E2 27047.245} C_VEL
LIN {X 0,Y 616.185,Z 728.776,A -85,B 0,C 180,E1 27046.702,E2 27046.702} C_VEL
LIN {X 0,Y 617.15,Z 706.897,A -85,B 0,C 180,E1 27046.325,E2 27046.325} C_VEL
LIN {X 0,Y 622.808,Z 466.074,A -85,B 0,C 180,E1 27043.067,E2 27043.067} C_VEL
LIN {X 0,Y 625.943,Z 335.01,A -85,B 0,C 180,E1 27041.249,E2 27041.249} C_VEL
LIN {X 0,Y 612.85,Z 314.28,A -85,B 0,C 180,E1 27039.577,E2 27039.577} C_VEL
LIN {X 0,Y 603.221,Z 300.406,A -85,B 0,C 180,E1 27038.282,E2 27038.282} C_VEL
LIN {X 0,Y 595.911,Z 290.208,A -85,B 0,C 180,E1 27037.251,E2 27037.251} C_VEL
LIN {X 0,Y 587.734,Z 278.902,A -85,B 0,C 180,E1 27036,E2 27036} C_VEL
LIN {X 0,Y 586.389,Z 276.39,A -85,B 0,C 180,E1 27035.554,E2 27035.554} C_VEL
LIN {X 0,Y 585.214,Z 273.22,A -85,B 0,C 180,E1 27034.96,E2 27034.96} C_VEL
LIN {X 0,Y 585.217,Z 273.072,A -85,B 0,C 180,E1 27031.752,E2 27031.752} C_VEL
LIN {X 0,Y 585.192,Z 273.083,A -85,B 0,C 180,E1 27028.918,E2 27028.918} C_VEL
LIN {X 0,Y 585.217,Z 273.031,A -85,B 0,C 180,E1 27025.721,E2 27025.721} C_VEL
LIN {X 0,Y 585.197,Z 273.087,A -85,B 0,C 180,E1 27022.715,E2 27022.715} C_VEL
LIN {X 0,Y 585.196,Z 273.035,A -85,B 0,C 180,E1 27019.359,E2 27019.359} C_VEL
LIN {X 0,Y 585.214,Z 273.082,A -85,B 0,C 180,E1 27016.375,E2 27016.375} C_VEL
LIN {X 0,Y 585.186,Z 273.032,A -85,B 0,C 180,E1 27013.11,E2 27013.11} C_VEL
LIN {X 0,Y 585.24,Z 273.08,A -85,B 0,C 180,E1 27010.036,E2 27010.036} C_VEL
LIN {X 0,Y 585.179,Z 273.022,A -85,B 0,C 180,E1 27006.87,E2 27006.87} C_VEL
LIN {X 0,Y 585.249,Z 273.078,A -85,B 0,C 180,E1 27003.821,E2 27003.821} C_VEL
LIN {X 0,Y 585.18,Z 273.031,A -85,B 0,C 180,E1 27000.685,E2 27000.685} C_VEL
LIN {X 0,Y 585.253,Z 273.064,A -85,B 0,C 180,E1 26997.65,E2 26997.65} C_VEL
LIN {X 0,Y 585.184,Z 273.049,A -85,B 0,C 180,E1 26994.509,E2 26994.509} C_VEL
LIN {X 0,Y 585.244,Z 273.041,A -85,B 0,C 180,E1 26991.353,E2 26991.353} C_VEL
LIN {X 0,Y 585.189,Z 273.065,A -85,B 0,C 180,E1 26988.268,E2 26988.268} C_VEL
LIN {X 0,Y 585.22,Z 273.033,A -85,B 0,C 180,E1 26985.049,E2 26985.049} C_VEL
LIN {X 0,Y 585.195,Z 273.077,A -85,B 0,C 180,E1 26982.088,E2 26982.088} C_VEL
LIN {X 0,Y 585.202,Z 273.037,A -85,B 0,C 180,E1 26978.763,E2 26978.763} C_VEL
LIN {X 0,Y 585.2,Z 273.08,A -85,B 0,C 180,E1 26975.898,E2 26975.898} C_VEL
LIN {X 0,Y 585.2,Z 273.079,A -85,B 0,C 180,E1 26972.527,E2 26972.527} C_VEL
LIN {X 0,Y 585.216,Z 273.077,A -85,B 0,C 180,E1 26969.619,E2 26969.619} C_VEL
LIN {X 0,Y 585.187,Z 273.028,A -85,B 0,C 180,E1 26966.317,E2 26966.317} C_VEL
LIN {X 0,Y 585.239,Z 273.037,A -85,B 0,C 180,E1 26963.253,E2 26963.253} C_VEL
LIN {X 0,Y 585.291,Z 273.498,A -85,B 0,C 180,E1 26962.665,E2 26962.665} C_VEL
LIN {X 0,Y 586.86,Z 277.035,A -85,B 0,C 180,E1 26962.043,E2 26962.043} C_VEL
LIN {X 0,Y 589.724,Z 283.018,A -85,B 0,C 180,E1 26961.02,E2 26961.02} C_VEL
LIN {X 0,Y 591.689,Z 286.871,A -85,B 0,C 180,E1 26960.425,E2 26960.425} C_VEL
LIN {X 0,Y 605.624,Z 306.533,A -85,B 0,C 180,E1 26958.432,E2 26958.432} C_VEL
LIN {X 0,Y 617.104,Z 323.965,A -85,B 0,C 180,E1 26956.909,E2 26956.909} C_VEL
LIN {X 0,Y 626.127,Z 338.813,A -85,B 0,C 180,E1 26955.764,E2 26955.764} C_VEL
LIN {X 0,Y 620.379,Z 573.672,A -85,B 0,C 180,E1 26952.553,E2 26952.553} C_VEL
LIN {X 0,Y 616.921,Z 720.786,A -85,B 0,C 180,E1 26950.563,E2 26950.563} C_VEL
LIN {X 0,Y 615.54,Z 748.126,A -85,B 0,C 180,E1 26950.045,E2 26950.045} C_VEL
LIN {X 0,Y 613.983,Z 770.909,A -85,B 0,C 180,E1 26949.456,E2 26949.456} C_VEL
LIN {X 0,Y 612.269,Z 792.237,A -85,B 0,C 180,E1 26948.777,E2 26948.777} C_VEL
LIN {X 0,Y 609.878,Z 818.259,A -85,B 0,C 180,E1 26947.759,E2 26947.759} C_VEL
LIN {X 0,Y 607.688,Z 838.898,A -85,B 0,C 180,E1 26946.793,E2 26946.793} C_VEL
LIN {X 0,Y 605.538,Z 857.93,A -85,B 0,C 180,E1 26945.77,E2 26945.77} C_VEL
LIN {X 0,Y 602.862,Z 880.5,A -85,B 0,C 180,E1 26944.384,E2 26944.384} C_VEL
LIN {X 0,Y 600.179,Z 901.279,A -85,B 0,C 180,E1 26942.896,E2 26942.896} C_VEL
LIN {X 0,Y 597.871,Z 919.154,A -85,B 0,C 180,E1 26941.452,E2 26941.452} C_VEL
LIN {X 0,Y 595.351,Z 938.977,A -85,B 0,C 180,E1 26939.644,E2 26939.644} C_VEL
LIN {X 0,Y 593.034,Z 956.692,A -85,B 0,C 180,E1 26937.787,E2 26937.787} C_VEL
LIN {X 0,Y 591.215,Z 971.238,A -85,B 0,C 180,E1 26936.086,E2 26936.086} C_VEL
LIN {X 0,Y 589.236,Z 988.389,A -85,B 0,C 180,E1 26933.82,E2 26933.82} C_VEL
LIN {X 0,Y 587.728,Z 1002.121,A -85,B 0,C 180,E1 26931.735,E2 26931.735} C_VEL
LIN {X 0,Y 586.559,Z 1014.451,A -85,B 0,C 180,E1 26929.622,E2 26929.622} C_VEL
LIN {X 0,Y 585.53,Z 1026.724,A -85,B 0,C 180,E1 26927.183,E2 26927.183} C_VEL
LIN {X 0,Y 584.908,Z 1035.88,A -85,B 0,C 180,E1 26925.061,E2 26925.061} C_VEL
LIN {X 0,Y 584.445,Z 1044.278,A -85,B 0,C 180,E1 26922.791,E2 26922.791} C_VEL
LIN {X 0,Y 584.131,Z 1051.878,A -85,B 0,C 180,E1 26920.255,E2 26920.255} C_VEL
LIN {X 0,Y 584.002,Z 1056.828,A -85,B 0,C 180,E1 26918.17,E2 26918.17} C_VEL
LIN {X 0,Y 583.942,Z 1060.486,A -85,B 0,C 180,E1 26916.193,E2 26916.193} C_VEL
LIN {X 0,Y 583.915,Z 1063.469,A -85,B 0,C 180,E1 26913.928,E2 26913.928} C_VEL
LIN {X 0,Y 583.903,Z 1065.191,A -85,B 0,C 180,E1 26911.374,E2 26911.374} C_VEL
LIN {X 0,Y 583.9,Z 1065.327,A -85,B 0,C 180,E1 26909.215,E2 26909.215} C_VEL
LIN {X 0,Y 583.913,Z 1064.369,A -85,B 0,C 180,E1 26907.154,E2 26907.154} C_VEL
LIN {X 0,Y 583.923,Z 1061.993,A -85,B 0,C 180,E1 26904.793,E2 26904.793} C_VEL
LIN {X 0,Y 583.995,Z 1057.654,A -85,B 0,C 180,E1 26902.226,E2 26902.226} C_VEL
LIN {X 0,Y 584.088,Z 1052.895,A -85,B 0,C 180,E1 26900.143,E2 26900.143} C_VEL
LIN {X 0,Y 584.326,Z 1046.968,A -85,B 0,C 180,E1 26898.05,E2 26898.05} C_VEL
LIN {X 0,Y 584.788,Z 1037.904,A -85,B 0,C 180,E1 26895.443,E2 26895.443} C_VEL
LIN {X 0,Y 585.389,Z 1028.563,A -85,B 0,C 180,E1 26893.222,E2 26893.222} C_VEL
LIN {X 0,Y 586.22,Z 1018.238,A -85,B 0,C 180,E1 26891.091,E2 26891.091} C_VEL
LIN {X 0,Y 587.554,Z 1004.03,A -85,B 0,C 180,E1 26888.573,E2 26888.573} C_VEL
LIN {X 0,Y 588.891,Z 991.192,A -85,B 0,C 180,E1 26886.59,E2 26886.59} C_VEL
LIN {X 0,Y 590.753,Z 975.45,A -85,B 0,C 180,E1 26884.431,E2 26884.431} C_VEL
LIN {X 0,Y 592.856,Z 958.082,A -85,B 0,C 180,E1 26882.367,E2 26882.367} C_VEL
LIN {X 0,Y 594.856,Z 942.526,A -85,B 0,C 180,E1 26880.716,E2 26880.716} C_VEL
LIN {X 0,Y 597.437,Z 922.816,A -85,B 0,C 180,E1 26878.859,E2 26878.859} C_VEL
LIN {X 0,Y 599.89,Z 903.466,A -85,B 0,C 180,E1 26877.272,E2 26877.272} C_VEL
LIN {X 0,Y 602.237,Z 884.996,A -85,B 0,C 180,E1 26875.926,E2 26875.926} C_VEL
LIN {X 0,Y 605.136,Z 861.553,A -85,B 0,C 180,E1 26874.435,E2 26874.435} C_VEL
LIN {X 0,Y 607.473,Z 840.935,A -85,B 0,C 180,E1 26873.31,E2 26873.31} C_VEL
LIN {X 0,Y 609.483,Z 822.054,A -85,B 0,C 180,E1 26872.41,E2 26872.41} C_VEL
LIN {X 0,Y 611.704,Z 799.428,A -85,B 0,C 180,E1 26871.481,E2 26871.481} C_VEL
LIN {X 0,Y 613.771,Z 774.114,A -85,B 0,C 180,E1 26870.638,E2 26870.638} C_VEL
LIN {X 0,Y 615.23,Z 753.257,A -85,B 0,C 180,E1 26870.079,E2 26870.079} C_VEL
LIN {X 0,Y 616.391,Z 733.147,A -85,B 0,C 180,E1 26869.651,E2 26869.651} C_VEL
LIN {X 0,Y 617.435,Z 705.256,A -85,B 0,C 180,E1 26869.211,E2 26869.211} C_VEL
LIN {X 0,Y 622.712,Z 468.147,A -85,B 0,C 180,E1 26866.03,E2 26866.03} C_VEL
LIN {X 0,Y 625.657,Z 338.336,A -85,B 0,C 180,E1 26864.252,E2 26864.252} C_VEL
LIN {X 0,Y 610.544,Z 314.865,A -85,B 0,C 180,E1 26862.434,E2 26862.434} C_VEL
LIN {X 0,Y 599.474,Z 298.413,A -85,B 0,C 180,E1 26861.021,E2 26861.021} C_VEL
LIN {X 0,Y 591.133,Z 286.262,A -85,B 0,C 180,E1 26859.872,E2 26859.872} C_VEL
LIN {X 0,Y 586.465,Z 276.469,A -85,B 0,C 180,E1 26858.347,E2 26858.347} C_VEL
LIN {X 0,Y 585.211,Z 273.222,A -85,B 0,C 180,E1 26857.806,E2 26857.806} C_VEL
LIN {X 0,Y 585.234,Z 273.034,A -85,B 0,C 180,E1 26854.677,E2 26854.677} C_VEL
LIN {X 0,Y 585.194,Z 273.086,A -85,B 0,C 180,E1 26851.638,E2 26851.638} C_VEL
LIN {X 0,Y 585.212,Z 273.031,A -85,B 0,C 180,E1 26848.367,E2 26848.367} C_VEL
LIN {X 0,Y 585.202,Z 273.085,A -85,B 0,C 180,E1 26845.396,E2 26845.396} C_VEL
LIN {X 0,Y 585.201,Z 273.086,A -85,B 0,C 180,E1 26842.08,E2 26842.08} C_VEL
LIN {X 0,Y 585.214,Z 273.077,A -85,B 0,C 180,E1 26839.119,E2 26839.119} C_VEL
LIN {X 0,Y 585.192,Z 273.075,A -85,B 0,C 180,E1 26835.853,E2 26835.853} C_VEL
LIN {X 0,Y 585.223,Z 273.068,A -85,B 0,C 180,E1 26832.934,E2 26832.934} C_VEL
LIN {X 0,Y 585.191,Z 273.08,A -85,B 0,C 180,E1 26829.739,E2 26829.739} C_VEL
LIN {X 0,Y 585.229,Z 273.077,A -85,B 0,C 180,E1 26826.77,E2 26826.77} C_VEL
LIN {X 0,Y 585.19,Z 273.072,A -85,B 0,C 180,E1 26823.625,E2 26823.625} C_VEL
LIN {X 0,Y 585.24,Z 273.068,A -85,B 0,C 180,E1 26820.587,E2 26820.587} C_VEL
LIN {X 0,Y 585.189,Z 273.084,A -85,B 0,C 180,E1 26817.454,E2 26817.454} C_VEL
LIN {X 0,Y 585.257,Z 273.069,A -85,B 0,C 180,E1 26814.313,E2 26814.313} C_VEL
LIN {X 0,Y 585.185,Z 273.066,A -85,B 0,C 180,E1 26811.253,E2 26811.253} C_VEL
LIN {X 0,Y 585.254,Z 273.07,A -85,B 0,C 180,E1 26808.169,E2 26808.169} C_VEL
LIN {X 0,Y 585.187,Z 273.085,A -85,B 0,C 180,E1 26805.048,E2 26805.048} C_VEL
LIN {X 0,Y 585.245,Z 273.071,A -85,B 0,C 180,E1 26801.884,E2 26801.884} C_VEL
LIN {X 0,Y 585.186,Z 273.068,A -85,B 0,C 180,E1 26798.867,E2 26798.867} C_VEL
LIN {X 0,Y 585.245,Z 273.056,A -85,B 0,C 180,E1 26795.793,E2 26795.793} C_VEL
LIN {X 0,Y 585.184,Z 273.023,A -85,B 0,C 180,E1 26792.686,E2 26792.686} C_VEL
LIN {X 0,Y 585.218,Z 273.075,A -85,B 0,C 180,E1 26789.442,E2 26789.442} C_VEL
LIN {X 0,Y 585.195,Z 273.019,A -85,B 0,C 180,E1 26786.385,E2 26786.385} C_VEL
LIN {X 0,Y 585.196,Z 273.074,A -85,B 0,C 180,E1 26783.096,E2 26783.096} C_VEL
LIN {X 0,Y 585.204,Z 273.084,A -85,B 0,C 180,E1 26780.253,E2 26780.253} C_VEL
LIN {X 0,Y 585.224,Z 273.309,A -85,B 0,C 180,E1 26778.389,E2 26778.389} C_VEL
LIN {X 0,Y 586.649,Z 276.712,A -85,B 0,C 180,E1 26777.814,E2 26777.814} C_VEL
LIN {X 0,Y 588.297,Z 280.114,A -85,B 0,C 180,E1 26777.35,E2 26777.35} C_VEL
LIN {X 0,Y 597.684,Z 293.174,A -85,B 0,C 180,E1 26776.08,E2 26776.08} C_VEL
LIN {X 0,Y 609.18,Z 309.804,A -85,B 0,C 180,E1 26774.606,E2 26774.606} C_VEL
LIN {X 0,Y 625.226,Z 334.354,A -85,B 0,C 180,E1 26772.671,E2 26772.671} C_VEL
LIN {X 0,Y 625.696,Z 335.681,A -85,B 0,C 180,E1 26772.607,E2 26772.607} C_VEL
LIN {X 0,Y 622.547,Z 470.61,A -85,B 0,C 180,E1 26770.767,E2 26770.767} C_VEL
LIN {X 0,Y 621.651,Z 478.309,A -85,B 0,C 180,E1 26770.726,E2 26770.726} C_VEL
LIN {X 0,Y 616.602,Z 498.912,A -85,B 0,C 180,E1 26770.845,E2 26770.845} C_VEL
LIN {X 0,Y 615.891,Z 505.521,A -85,B 0,C 180,E1 26770.804,E2 26770.804} C_VEL
LIN {X 0,Y 610.932,Z 710.903,A -85,B 0,C 180,E1 26768.015,E2 26768.015} C_VEL
LIN {X 0,Y 609.594,Z 737.261,A -85,B 0,C 180,E1 26767.524,E2 26767.524} C_VEL
LIN {X 0,Y 607.889,Z 761.273,A -85,B 0,C 180,E1 26766.903,E2 26766.903} C_VEL
LIN {X 0,Y 606.11,Z 782.432,A -85,B 0,C 180,E1 26766.225,E2 26766.225} C_VEL
LIN {X 0,Y 603.731,Z 807.37,A -85,B 0,C 180,E1 26765.252,E2 26765.252} C_VEL
LIN {X 0,Y 601.35,Z 828.645,A -85,B 0,C 180,E1 26764.252,E2 26764.252} C_VEL
LIN {X 0,Y 599.015,Z 848.143,A -85,B 0,C 180,E1 26763.196,E2 26763.196} C_VEL
LIN {X 0,Y 596.249,Z 870.166,A -85,B 0,C 180,E1 26761.83,E2 26761.83} C_VEL
LIN {X 0,Y 593.267,Z 891.804,A -85,B 0,C 180,E1 26760.26,E2 26760.26} C_VEL
LIN {X 0,Y 590.858,Z 909.185,A -85,B 0,C 180,E1 26758.835,E2 26758.835} C_VEL
LIN {X 0,Y 588.137,Z 929.06,A -85,B 0,C 180,E1 26756.996,E2 26756.996} C_VEL
LIN {X 0,Y 585.724,Z 946.4,A -85,B 0,C 180,E1 26755.155,E2 26755.155} C_VEL
LIN {X 0,Y 583.772,Z 961.125,A -85,B 0,C 180,E1 26753.414,E2 26753.414} C_VEL
LIN {X 0,Y 581.681,Z 978.021,A -85,B 0,C 180,E1 26751.16,E2 26751.16} C_VEL
LIN {X 0,Y 580.106,Z 991.374,A -85,B 0,C 180,E1 26749.116,E2 26749.116} C_VEL
LIN {X 0,Y 578.889,Z 1003.218,A -85,B 0,C 180,E1 26747.075,E2 26747.075} C_VEL
LIN {X 0,Y 577.728,Z 1016.037,A -85,B 0,C 180,E1 26744.534,E2 26744.534} C_VEL
LIN {X 0,Y 577.003,Z 1025.565,A -85,B 0,C 180,E1 26742.307,E2 26742.307} C_VEL
LIN {X 0,Y 576.537,Z 1033.361,A -85,B 0,C 180,E1 26740.189,E2 26740.189} C_VEL
LIN {X 0,Y 576.19,Z 1041.307,A -85,B 0,C 180,E1 26737.579,E2 26737.579} C_VEL
LIN {X 0,Y 576.011,Z 1046.746,A -85,B 0,C 180,E1 26735.279,E2 26735.279} C_VEL
LIN {X 0,Y 575.942,Z 1050.564,A -85,B 0,C 180,E1 26733.185,E2 26733.185} C_VEL
LIN {X 0,Y 575.92,Z 1053.629,A -85,B 0,C 180,E1 26730.796,E2 26730.796} C_VEL
LIN {X 0,Y 575.908,Z 1055.222,A -85,B 0,C 180,E1 26728.209,E2 26728.209} C_VEL
LIN {X 0,Y 575.902,Z 1055.317,A -85,B 0,C 180,E1 26726.117,E2 26726.117} C_VEL
LIN {X 0,Y 575.916,Z 1054.336,A -85,B 0,C 180,E1 26724.021,E2 26724.021} C_VEL
LIN {X 0,Y 575.921,Z 1051.924,A -85,B 0,C 180,E1 26721.614,E2 26721.614} C_VEL
LIN {X 0,Y 575.995,Z 1047.696,A -85,B 0,C 180,E1 26719.093,E2 26719.093} C_VEL
LIN {X 0,Y 576.107,Z 1042.895,A -85,B 0,C 180,E1 26716.96,E2 26716.96} C_VEL
LIN {X 0,Y 576.361,Z 1036.897,A -85,B 0,C 180,E1 26714.814,E2 26714.814} C_VEL
LIN {X 0,Y 576.883,Z 1027.669,A -85,B 0,C 180,E1 26712.134,E2 26712.134} C_VEL
LIN {X 0,Y 577.507,Z 1018.604,A -85,B 0,C 180,E1 26709.952,E2 26709.952} C_VEL
LIN {X 0,Y 578.366,Z 1008.626,A -85,B 0,C 180,E1 26707.859,E2 26707.859} C_VEL
LIN {X 0,Y 579.768,Z 994.661,A -85,B 0,C 180,E1 26705.332,E2 26705.332} C_VEL
LIN {X 0,Y 581.189,Z 981.859,A -85,B 0,C 180,E1 26703.319,E2 26703.319} C_VEL
LIN {X 0,Y 583.08,Z 966.686,A -85,B 0,C 180,E1 26701.198,E2 26701.198} C_VEL
LIN {X 0,Y 585.358,Z 949.095,A -85,B 0,C 180,E1 26699.059,E2 26699.059} C_VEL
LIN {X 0,Y 587.561,Z 932.995,A -85,B 0,C 180,E1 26697.32,E2 26697.32} C_VEL
LIN {X 0,Y 590.325,Z 913.308,A -85,B 0,C 180,E1 26695.43,E2 26695.43} C_VEL
LIN {X 0,Y 592.942,Z 894.116,A -85,B 0,C 180,E1 26693.828,E2 26693.828} C_VEL
LIN {X 0,Y 595.489,Z 875.437,A -85,B 0,C 180,E1 26692.446,E2 26692.446} C_VEL
LIN {X 0,Y 598.514,Z 852.462,A -85,B 0,C 180,E1 26690.963,E2 26690.963} C_VEL
LIN {X 0,Y 601.042,Z 831.394,A -85,B 0,C 180,E1 26689.799,E2 26689.799} C_VEL
LIN {X 0,Y 603.134,Z 812.818,A -85,B 0,C 180,E1 26688.904,E2 26688.904} C_VEL
LIN {X 0,Y 605.415,Z 790.745,A -85,B 0,C 180,E1 26687.987,E2 26687.987} C_VEL
LIN {X 0,Y 607.618,Z 765.116,A -85,B 0,C 180,E1 26687.121,E2 26687.121} C_VEL
LIN {X 0,Y 609.157,Z 744.044,A -85,B 0,C 180,E1 26686.551,E2 26686.551} C_VEL
LIN {X 0,Y 610.376,Z 723.732,A -85,B 0,C 180,E1 26686.116,E2 26686.116} C_VEL
LIN {X 0,Y 611.487,Z 694.666,A -85,B 0,C 180,E1 26685.657,E2 26685.657} C_VEL
LIN {X 0,Y 617.303,Z 458.403,A -85,B 0,C 180,E1 26682.436,E2 26682.436} C_VEL
LIN {X 0,Y 620.319,Z 338.523,A -85,B 0,C 180,E1 26680.755,E2 26680.755} C_VEL
LIN {X 0,Y 608.163,Z 319.331,A -85,B 0,C 180,E1 26679.165,E2 26679.165} C_VEL
LIN {X 0,Y 596.891,Z 302.9,A -85,B 0,C 180,E1 26677.603,E2 26677.603} C_VEL
LIN {X 0,Y 585.874,Z 287.864,A -85,B 0,C 180,E1 26675.981,E2 26675.981} C_VEL
LIN {X 0,Y 582.108,Z 282.971,A -85,B 0,C 180,E1 26675.401,E2 26675.401} C_VEL
LIN {X 0,Y 579.377,Z 278.74,A -85,B 0,C 180,E1 26674.897,E2 26674.897} C_VEL
LIN {X 0,Y 577.41,Z 274.65,A -85,B 0,C 180,E1 26674.13,E2 26674.13} C_VEL
LIN {X 0,Y 577.296,Z 274.103,A -85,B 0,C 180,E1 26673.898,E2 26673.898} C_VEL
LIN {X 0,Y 577.253,Z 274.046,A -85,B 0,C 180,E1 26670.845,E2 26670.845} C_VEL
LIN {X 0,Y 577.262,Z 274.053,A -85,B 0,C 180,E1 26667.521,E2 26667.521} C_VEL
LIN {X 0,Y 577.277,Z 274.036,A -85,B 0,C 180,E1 26664.454,E2 26664.454} C_VEL
LIN {X 0,Y 577.249,Z 274.035,A -85,B 0,C 180,E1 26661.225,E2 26661.225} C_VEL
LIN {X 0,Y 577.3,Z 274.047,A -85,B 0,C 180,E1 26658.166,E2 26658.166} C_VEL
LIN {X 0,Y 577.246,Z 274.036,A -85,B 0,C 180,E1 26655.06,E2 26655.06} C_VEL
LIN {X 0,Y 577.305,Z 274.037,A -85,B 0,C 180,E1 26651.996,E2 26651.996} C_VEL
LIN {X 0,Y 577.246,Z 274.047,A -85,B 0,C 180,E1 26648.868,E2 26648.868} C_VEL
LIN {X 0,Y 577.313,Z 274.015,A -85,B 0,C 180,E1 26645.765,E2 26645.765} C_VEL
LIN {X 0,Y 577.248,Z 274.067,A -85,B 0,C 180,E1 26642.581,E2 26642.581} C_VEL
LIN {X 0,Y 577.294,Z 274.01,A -85,B 0,C 180,E1 26639.405,E2 26639.405} C_VEL
LIN {X 0,Y 577.256,Z 274.075,A -85,B 0,C 180,E1 26636.325,E2 26636.325} C_VEL
LIN {X 0,Y 577.258,Z 274.007,A -85,B 0,C 180,E1 26632.982,E2 26632.982} C_VEL
LIN {X 0,Y 577.268,Z 274.066,A -85,B 0,C 180,E1 26630.025,E2 26630.025} C_VEL
LIN {X 0,Y 577.248,Z 274.012,A -85,B 0,C 180,E1 26626.681,E2 26626.681} C_VEL
LIN {X 0,Y 577.296,Z 274.058,A -85,B 0,C 180,E1 26623.645,E2 26623.645} C_VEL
LIN {X 0,Y 577.246,Z 274.022,A -85,B 0,C 180,E1 26620.441,E2 26620.441} C_VEL
LIN {X 0,Y 577.325,Z 274.059,A -85,B 0,C 180,E1 26617.28,E2 26617.28} C_VEL
LIN {X 0,Y 577.251,Z 274.066,A -85,B 0,C 180,E1 26614.119,E2 26614.119} C_VEL
LIN {X 0,Y 577.31,Z 274.058,A -85,B 0,C 180,E1 26610.99,E2 26610.99} C_VEL
LIN {X 0,Y 577.243,Z 274.015,A -85,B 0,C 180,E1 26607.991,E2 26607.991} C_VEL
LIN {X 0,Y 577.293,Z 274.062,A -85,B 0,C 180,E1 26604.776,E2 26604.776} C_VEL
LIN {X 0,Y 577.297,Z 274.304,A -85,B 0,C 180,E1 26603.676,E2 26603.676} C_VEL
LIN {X 0,Y 578.743,Z 277.68,A -85,B 0,C 180,E1 26603.041,E2 26603.041} C_VEL
LIN {X 0,Y 583.132,Z 286.505,A -85,B 0,C 180,E1 26601.506,E2 26601.506} C_VEL
LIN {X 0,Y 595.044,Z 303.029,A -85,B 0,C 180,E1 26599.706,E2 26599.706} C_VEL
LIN {X 0,Y 605.592,Z 318.434,A -85,B 0,C 180,E1 26598.224,E2 26598.224} C_VEL
LIN {X 0,Y 616.638,Z 335.732,A -85,B 0,C 180,E1 26596.757,E2 26596.757} C_VEL
LIN {X 0,Y 620.529,Z 342.444,A -85,B 0,C 180,E1 26596.252,E2 26596.252} C_VEL
LIN {X 0,Y 614.462,Z 576.437,A -85,B 0,C 180,E1 26593.026,E2 26593.026} C_VEL
LIN {X 0,Y 610.853,Z 720.678,A -85,B 0,C 180,E1 26591.054,E2 26591.054} C_VEL
LIN {X 0,Y 609.396,Z 747.974,A -85,B 0,C 180,E1 26590.535,E2 26590.535} C_VEL
LIN {X 0,Y 607.733,Z 771.143,A -85,B 0,C 180,E1 26589.931,E2 26589.931} C_VEL
LIN {X 0,Y 605.9,Z 792.884,A -85,B 0,C 180,E1 26589.232,E2 26589.232} C_VEL
LIN {X 0,Y 603.324,Z 819.302,A -85,B 0,C 180,E1 26588.183,E2 26588.183} C_VEL
LIN {X 0,Y 601.147,Z 838.808,A -85,B 0,C 180,E1 26587.26,E2 26587.26} C_VEL
LIN {X 0,Y 598.884,Z 857.841,A -85,B 0,C 180,E1 26586.23,E2 26586.23} C_VEL
LIN {X 0,Y 596.071,Z 880.412,A -85,B 0,C 180,E1 26584.832,E2 26584.832} C_VEL
LIN {X 0,Y 593.246,Z 901.191,A -85,B 0,C 180,E1 26583.33,E2 26583.33} C_VEL
LIN {X 0,Y 590.847,Z 918.72,A -85,B 0,C 180,E1 26581.902,E2 26581.902} C_VEL
LIN {X 0,Y 588.177,Z 938.555,A -85,B 0,C 180,E1 26580.084,E2 26580.084} C_VEL
LIN {X 0,Y 585.748,Z 956.227,A -85,B 0,C 180,E1 26578.219,E2 26578.219} C_VEL
LIN {X 0,Y 583.756,Z 971.237,A -85,B 0,C 180,E1 26576.445,E2 26576.445} C_VEL
LIN {X 0,Y 581.725,Z 987.686,A -85,B 0,C 180,E1 26574.255,E2 26574.255} C_VEL
LIN {X 0,Y 580.117,Z 1001.276,A -85,B 0,C 180,E1 26572.177,E2 26572.177} C_VEL
LIN {X 0,Y 578.931,Z 1012.73,A -85,B 0,C 180,E1 26570.208,E2 26570.208} C_VEL
LIN {X 0,Y 577.788,Z 1025.34,A -85,B 0,C 180,E1 26567.733,E2 26567.733} C_VEL
LIN {X 0,Y 577.033,Z 1035.068,A -85,B 0,C 180,E1 26565.477,E2 26565.477} C_VEL
LIN {X 0,Y 576.565,Z 1042.894,A -85,B 0,C 180,E1 26563.369,E2 26563.369} C_VEL
LIN {X 0,Y 576.201,Z 1050.79,A -85,B 0,C 180,E1 26560.829,E2 26560.829} C_VEL
LIN {X 0,Y 576.014,Z 1056.621,A -85,B 0,C 180,E1 26558.384,E2 26558.384} C_VEL
LIN {X 0,Y 575.949,Z 1060.326,A -85,B 0,C 180,E1 26556.379,E2 26556.379} C_VEL
LIN {X 0,Y 575.908,Z 1063.13,A -85,B 0,C 180,E1 26554.281,E2 26554.281} C_VEL
LIN {X 0,Y 575.9,Z 1065.099,A -85,B 0,C 180,E1 26551.791,E2 26551.791} C_VEL
LIN {X 0,Y 575.895,Z 1065.372,A -85,B 0,C 180,E1 26549.403,E2 26549.403} C_VEL
LIN {X 0,Y 575.913,Z 1064.505,A -85,B 0,C 180,E1 26547.313,E2 26547.313} C_VEL
LIN {X 0,Y 575.908,Z 1062.561,A -85,B 0,C 180,E1 26545.22,E2 26545.22} C_VEL
LIN {X 0,Y 575.98,Z 1058.884,A -85,B 0,C 180,E1 26542.72,E2 26542.72} C_VEL
LIN {X 0,Y 576.091,Z 1053.403,A -85,B 0,C 180,E1 26540.207,E2 26540.207} C_VEL
LIN {X 0,Y 576.333,Z 1047.609,A -85,B 0,C 180,E1 26538.097,E2 26538.097} C_VEL
LIN {X 0,Y 576.749,Z 1039.745,A -85,B 0,C 180,E1 26535.725,E2 26535.725} C_VEL
LIN {X 0,Y 577.442,Z 1029.479,A -85,B 0,C 180,E1 26533.192,E2 26533.192} C_VEL
LIN {X 0,Y 578.261,Z 1019.781,A -85,B 0,C 180,E1 26531.135,E2 26531.135} C_VEL
LIN {X 0,Y 579.546,Z 1006.984,A -85,B 0,C 180,E1 26528.758,E2 26528.758} C_VEL
LIN {X 0,Y 581.101,Z 992.591,A -85,B 0,C 180,E1 26526.472,E2 26526.472} C_VEL
LIN {X 0,Y 582.74,Z 979.314,A -85,B 0,C 180,E1 26524.599,E2 26524.599} C_VEL
LIN {X 0,Y 585.011,Z 961.783,A -85,B 0,C 180,E1 26522.407,E2 26522.407} C_VEL
LIN {X 0,Y 587.186,Z 945.545,A -85,B 0,C 180,E1 26520.632,E2 26520.632} C_VEL
LIN {X 0,Y 589.46,Z 928.994,A -85,B 0,C 180,E1 26519.015,E2 26519.015} C_VEL
LIN {X 0,Y 592.353,Z 907.893,A -85,B 0,C 180,E1 26517.191,E2 26517.191} C_VEL
LIN {X 0,Y 594.923,Z 888.523,A -85,B 0,C 180,E1 26515.734,E2 26515.734} C_VEL
LIN {X 0,Y 597.441,Z 869.293,A -85,B 0,C 180,E1 26514.454,E2 26514.454} C_VEL
LIN {X 0,Y 600.474,Z 844.879,A -85,B 0,C 180,E1 26513.05,E2 26513.05} C_VEL
LIN {X 0,Y 602.71,Z 824.994,A -85,B 0,C 180,E1 26512.073,E2 26512.073} C_VEL
LIN {X 0,Y 604.694,Z 805.776,A -85,B 0,C 180,E1 26511.254,E2 26511.254} C_VEL
LIN {X 0,Y 606.781,Z 783.432,A -85,B 0,C 180,E1 26510.446,E2 26510.446} C_VEL
LIN {X 0,Y 608.79,Z 757.536,A -85,B 0,C 180,E1 26509.699,E2 26509.699} C_VEL
LIN {X 0,Y 610.068,Z 736.891,A -85,B 0,C 180,E1 26509.236,E2 26509.236} C_VEL
LIN {X 0,Y 611.053,Z 715.114,A -85,B 0,C 180,E1 26508.863,E2 26508.863} C_VEL
LIN {X 0,Y 616.62,Z 480.135,A -85,B 0,C 180,E1 26505.682,E2 26505.682} C_VEL
LIN {X 0,Y 619.876,Z 341.829,A -85,B 0,C 180,E1 26503.773,E2 26503.773} C_VEL
LIN {X 0,Y 604.457,Z 317.847,A -85,B 0,C 180,E1 26501.872,E2 26501.872} C_VEL
LIN {X 0,Y 590.149,Z 296.72,A -85,B 0,C 180,E1 26499.984,E2 26499.984} C_VEL
LIN {X 0,Y 582.725,Z 286.046,A -85,B 0,C 180,E1 26498.904,E2 26498.904} C_VEL
LIN {X 0,Y 577.373,Z 274.436,A -85,B 0,C 180,E1 26497.012,E2 26497.012} C_VEL
LIN {X 0,Y 577.265,Z 274.078,A -85,B 0,C 180,E1 26496.327,E2 26496.327} C_VEL
LIN {X 0,Y 577.289,Z 274.023,A -85,B 0,C 180,E1 26493.184,E2 26493.184} C_VEL
LIN {X 0,Y 577.249,Z 274.04,A -85,B 0,C 180,E1 26489.994,E2 26489.994} C_VEL
LIN {X 0,Y 577.304,Z 274.041,A -85,B 0,C 180,E1 26486.987,E2 26486.987} C_VEL
LIN {X 0,Y 577.249,Z 274.058,A -85,B 0,C 180,E1 26483.803,E2 26483.803} C_VEL
LIN {X 0,Y 577.319,Z 274.053,A -85,B 0,C 180,E1 26480.691,E2 26480.691} C_VEL
LIN {X 0,Y 577.25,Z 274.07,A -85,B 0,C 180,E1 26477.542,E2 26477.542} C_VEL
LIN {X 0,Y 577.299,Z 274.071,A -85,B 0,C 180,E1 26474.34,E2 26474.34} C_VEL
LIN {X 0,Y 577.254,Z 274.069,A -85,B 0,C 180,E1 26471.288,E2 26471.288} C_VEL
LIN {X 0,Y 577.267,Z 274.057,A -85,B 0,C 180,E1 26467.965,E2 26467.965} C_VEL
LIN {X 0,Y 577.26,Z 274.065,A -85,B 0,C 180,E1 26465.068,E2 26465.068} C_VEL
LIN {X 0,Y 577.257,Z 274.072,A -85,B 0,C 180,E1 26461.687,E2 26461.687} C_VEL
LIN {X 0,Y 577.282,Z 274.061,A -85,B 0,C 180,E1 26458.71,E2 26458.71} C_VEL
LIN {X 0,Y 577.247,Z 274.055,A -85,B 0,C 180,E1 26455.43,E2 26455.43} C_VEL
LIN {X 0,Y 577.318,Z 274.057,A -85,B 0,C 180,E1 26452.336,E2 26452.336} C_VEL
LIN {X 0,Y 577.25,Z 274.074,A -85,B 0,C 180,E1 26449.117,E2 26449.117} C_VEL
LIN {X 0,Y 577.302,Z 274.06,A -85,B 0,C 180,E1 26445.91,E2 26445.91} C_VEL
LIN {X 0,Y 577.25,Z 274.053,A -85,B 0,C 180,E1 26442.874,E2 26442.874} C_VEL
LIN {X 0,Y 577.279,Z 274.055,A -85,B 0,C 180,E1 26439.626,E2 26439.626} C_VEL
LIN {X 0,Y 577.253,Z 274.073,A -85,B 0,C 180,E1 26436.738,E2 26436.738} C_VEL
LIN {X 0,Y 577.267,Z 273.998,A -85,B 0,C 180,E1 26433.456,E2 26433.456} C_VEL
LIN {X 0,Y 577.26,Z 274.072,A -85,B 0,C 180,E1 26430.533,E2 26430.533} C_VEL
LIN {X 0,Y 577.249,Z 274.005,A -85,B 0,C 180,E1 26427.15,E2 26427.15} C_VEL
LIN {X 0,Y 577.281,Z 274.072,A -85,B 0,C 180,E1 26424.155,E2 26424.155} C_VEL
LIN {X 0,Y 577.25,Z 274.07,A -85,B 0,C 180,E1 26420.896,E2 26420.896} C_VEL
LIN {X 0,Y 577.308,Z 274.308,A -85,B 0,C 180,E1 26419.235,E2 26419.235} C_VEL
LIN {X 0,Y 578.561,Z 277.564,A -85,B 0,C 180,E1 26418.686,E2 26418.686} C_VEL
LIN {X 0,Y 580.031,Z 280.288,A -85,B 0,C 180,E1 26418.303,E2 26418.303} C_VEL
LIN {X 0,Y 592.862,Z 297.894,A -85,B 0,C 180,E1 26416.519,E2 26416.519} C_VEL
LIN {X 0,Y 605.816,Z 317.02,A -85,B 0,C 180,E1 26414.822,E2 26414.822} C_VEL
LIN {X 0,Y 619.954,Z 338.69,A -85,B 0,C 180,E1 26413.09,E2 26413.09} C_VEL
LIN {X 0,Y 615.891,Z 505.521,A -85,B 0,C 180,E1 26410.804,E2 26410.804} C_VEL
LIN {X 0,Y 614.972,Z 513.22,A -85,B 0,C 180,E1 26410.763,E2 26410.763} C_VEL
LIN {X 0,Y 609.895,Z 533.813,A -85,B 0,C 180,E1 26410.885,E2 26410.885} C_VEL
LIN {X 0,Y 609.182,Z 540.418,A -85,B 0,C 180,E1 26410.843,E2 26410.843} C_VEL
LIN {X 0,Y 604.866,Z 711.321,A -85,B 0,C 180,E1 26408.505,E2 26408.505} C_VEL
LIN {X 0,Y 603.437,Z 738.054,A -85,B 0,C 180,E1 26408.001,E2 26408.001} C_VEL
LIN {X 0,Y 601.684,Z 761.77,A -85,B 0,C 180,E1 26407.382,E2 26407.382} C_VEL
LIN {X 0,Y 599.818,Z 783.039,A -85,B 0,C 180,E1 26406.695,E2 26406.695} C_VEL
LIN {X 0,Y 597.261,Z 808.391,A -85,B 0,C 180,E1 26405.692,E2 26405.692} C_VEL
LIN {X 0,Y 594.787,Z 829.468,A -85,B 0,C 180,E1 26404.689,E2 26404.689} C_VEL
LIN {X 0,Y 592.334,Z 848.977,A -85,B 0,C 180,E1 26403.62,E2 26403.62} C_VEL
LIN {X 0,Y 589.324,Z 871.613,A -85,B 0,C 180,E1 26402.192,E2 26402.192} C_VEL
LIN {X 0,Y 586.408,Z 891.796,A -85,B 0,C 180,E1 26400.709,E2 26400.709} C_VEL
LIN {X 0,Y 583.866,Z 909.187,A -85,B 0,C 180,E1 26399.27,E2 26399.27} C_VEL
LIN {X 0,Y 580.967,Z 929.077,A -85,B 0,C 180,E1 26397.412,E2 26397.412} C_VEL
LIN {X 0,Y 578.354,Z 946.855,A -85,B 0,C 180,E1 26395.498,E2 26395.498} C_VEL
LIN {X 0,Y 576.136,Z 962.574,A -85,B 0,C 180,E1 26393.601,E2 26393.601} C_VEL
LIN {X 0,Y 573.85,Z 979.893,A -85,B 0,C 180,E1 26391.219,E2 26391.219} C_VEL
LIN {X 0,Y 572.316,Z 992.273,A -85,B 0,C 180,E1 26389.281,E2 26389.281} C_VEL
LIN {X 0,Y 570.982,Z 1004.594,A -85,B 0,C 180,E1 26387.109,E2 26387.109} C_VEL
LIN {X 0,Y 569.77,Z 1017.139,A -85,B 0,C 180,E1 26384.534,E2 26384.534} C_VEL
LIN {X 0,Y 569.076,Z 1025.738,A -85,B 0,C 180,E1 26382.481,E2 26382.481} C_VEL
LIN {X 0,Y 568.564,Z 1033.861,A -85,B 0,C 180,E1 26380.231,E2 26380.231} C_VEL
LIN {X 0,Y 568.198,Z 1041.67,A -85,B 0,C 180,E1 26377.584,E2 26377.584} C_VEL
LIN {X 0,Y 568.016,Z 1046.834,A -85,B 0,C 180,E1 26375.353,E2 26375.353} C_VEL
LIN {X 0,Y 567.948,Z 1050.473,A -85,B 0,C 180,E1 26373.331,E2 26373.331} C_VEL
LIN {X 0,Y 567.918,Z 1053.452,A -85,B 0,C 180,E1 26371.009,E2 26371.009} C_VEL
LIN {X 0,Y 567.898,Z 1055.186,A -85,B 0,C 180,E1 26368.386,E2 26368.386} C_VEL
LIN {X 0,Y 567.899,Z 1055.33,A -85,B 0,C 180,E1 26366.164,E2 26366.164} C_VEL
LIN {X 0,Y 567.916,Z 1054.375,A -85,B 0,C 180,E1 26364.038,E2 26364.038} C_VEL
LIN {X 0,Y 567.925,Z 1052.104,A -85,B 0,C 180,E1 26361.699,E2 26361.699} C_VEL
LIN {X 0,Y 568,Z 1047.815,A -85,B 0,C 180,E1 26359.04,E2 26359.04} C_VEL
LIN {X 0,Y 568.122,Z 1043.041,A -85,B 0,C 180,E1 26356.877,E2 26356.877} C_VEL
LIN {X 0,Y 568.387,Z 1037.071,A -85,B 0,C 180,E1 26354.7,E2 26354.7} C_VEL
LIN {X 0,Y 568.923,Z 1028.311,A -85,B 0,C 180,E1 26352.088,E2 26352.088} C_VEL
LIN {X 0,Y 569.614,Z 1018.865,A -85,B 0,C 180,E1 26349.769,E2 26349.769} C_VEL
LIN {X 0,Y 570.527,Z 1008.918,A -85,B 0,C 180,E1 26347.647,E2 26347.647} C_VEL
LIN {X 0,Y 572.012,Z 995.021,A -85,B 0,C 180,E1 26345.085,E2 26345.085} C_VEL
LIN {X 0,Y 573.536,Z 982.256,A -85,B 0,C 180,E1 26343.046,E2 26343.046} C_VEL
LIN {X 0,Y 575.315,Z 968.659,A -85,B 0,C 180,E1 26341.108,E2 26341.108} C_VEL
LIN {X 0,Y 577.884,Z 950.141,A -85,B 0,C 180,E1 26338.788,E2 26338.788} C_VEL
LIN {X 0,Y 580.135,Z 934.598,A -85,B 0,C 180,E1 26337.074,E2 26337.074} C_VEL
LIN {X 0,Y 582.523,Z 918.471,A -85,B 0,C 180,E1 26335.479,E2 26335.479} C_VEL
LIN {X 0,Y 585.747,Z 896.324,A -85,B 0,C 180,E1 26333.555,E2 26333.555} C_VEL
LIN {X 0,Y 588.387,Z 877.861,A -85,B 0,C 180,E1 26332.159,E2 26332.159} C_VEL
LIN {X 0,Y 591.18,Z 857.869,A -85,B 0,C 180,E1 26330.823,E2 26330.823} C_VEL
LIN {X 0,Y 594.18,Z 834.695,A -85,B 0,C 180,E1 26329.492,E2 26329.492} C_VEL
LIN {X 0,Y 596.485,Z 815.255,A -85,B 0,C 180,E1 26328.531,E2 26328.531} C_VEL
LIN {X 0,Y 598.615,Z 795.616,A -85,B 0,C 180,E1 26327.69,E2 26327.69} C_VEL
LIN {X 0,Y 600.965,Z 771.686,A -85,B 0,C 180,E1 26326.824,E2 26326.824} C_VEL
LIN {X 0,Y 602.904,Z 746.763,A -85,B 0,C 180,E1 26326.118,E2 26326.118} C_VEL
LIN {X 0,Y 604.175,Z 727.036,A -85,B 0,C 180,E1 26325.677,E2 26325.677} C_VEL
LIN {X 0,Y 605.206,Z 704.901,A -85,B 0,C 180,E1 26325.298,E2 26325.298} C_VEL
LIN {X 0,Y 611.535,Z 464.605,A -85,B 0,C 180,E1 26321.987,E2 26321.987} C_VEL
LIN {X 0,Y 614.815,Z 342.158,A -85,B 0,C 180,E1 26320.261,E2 26320.261} C_VEL
LIN {X 0,Y 602.101,Z 322.111,A -85,B 0,C 180,E1 26318.548,E2 26318.548} C_VEL
LIN {X 0,Y 589.253,Z 303.656,A -85,B 0,C 180,E1 26316.707,E2 26316.707} C_VEL
LIN {X 0,Y 578.877,Z 289.684,A -85,B 0,C 180,E1 26315.113,E2 26315.113} C_VEL
LIN {X 0,Y 574.675,Z 284.169,A -85,B 0,C 180,E1 26314.436,E2 26314.436} C_VEL
LIN {X 0,Y 571.209,Z 279.277,A -85,B 0,C 180,E1 26313.825,E2 26313.825} C_VEL
LIN {X 0,Y 569.54,Z 276.202,A -85,B 0,C 180,E1 26313.213,E2 26313.213} C_VEL
LIN {X 0,Y 569.333,Z 275.199,A -85,B 0,C 180,E1 26312.986,E2 26312.986} C_VEL
LIN {X 0,Y 569.346,Z 275.032,A -85,B 0,C 180,E1 26309.802,E2 26309.802} C_VEL
LIN {X 0,Y 569.312,Z 275.019,A -85,B 0,C 180,E1 26306.832,E2 26306.832} C_VEL
LIN {X 0,Y 569.328,Z 275.055,A -85,B 0,C 180,E1 26303.495,E2 26303.495} C_VEL
LIN {X 0,Y 569.32,Z 275.007,A -85,B 0,C 180,E1 26300.564,E2 26300.564} C_VEL
LIN {X 0,Y 569.321,Z 275.063,A -85,B 0,C 180,E1 26297.266,E2 26297.266} C_VEL
LIN {X 0,Y 569.344,Z 275,A -85,B 0,C 180,E1 26294.205,E2 26294.205} C_VEL
LIN {X 0,Y 569.311,Z 275.061,A -85,B 0,C 180,E1 26290.934,E2 26290.934} C_VEL
LIN {X 0,Y 569.38,Z 274.992,A -85,B 0,C 180,E1 26287.771,E2 26287.771} C_VEL
LIN {X 0,Y 569.31,Z 275.051,A -85,B 0,C 180,E1 26284.634,E2 26284.634} C_VEL
LIN {X 0,Y 569.352,Z 275.013,A -85,B 0,C 180,E1 26281.409,E2 26281.409} C_VEL
LIN {X 0,Y 569.312,Z 275.026,A -85,B 0,C 180,E1 26278.39,E2 26278.39} C_VEL
LIN {X 0,Y 569.33,Z 275.04,A -85,B 0,C 180,E1 26275.063,E2 26275.063} C_VEL
LIN {X 0,Y 569.318,Z 275,A -85,B 0,C 180,E1 26272.115,E2 26272.115} C_VEL
LIN {X 0,Y 569.318,Z 275.054,A -85,B 0,C 180,E1 26268.758,E2 26268.758} C_VEL
LIN {X 0,Y 569.353,Z 274.993,A -85,B 0,C 180,E1 26265.663,E2 26265.663} C_VEL
LIN {X 0,Y 569.313,Z 275.06,A -85,B 0,C 180,E1 26262.491,E2 26262.491} C_VEL
LIN {X 0,Y 569.374,Z 274.995,A -85,B 0,C 180,E1 26259.33,E2 26259.33} C_VEL
LIN {X 0,Y 569.313,Z 275.064,A -85,B 0,C 180,E1 26256.174,E2 26256.174} C_VEL
LIN {X 0,Y 569.358,Z 275.057,A -85,B 0,C 180,E1 26252.92,E2 26252.92} C_VEL
LIN {X 0,Y 569.317,Z 275.067,A -85,B 0,C 180,E1 26249.964,E2 26249.964} C_VEL
LIN {X 0,Y 569.331,Z 274.992,A -85,B 0,C 180,E1 26246.653,E2 26246.653} C_VEL
LIN {X 0,Y 569.382,Z 275.327,A -85,B 0,C 180,E1 26244.676,E2 26244.676} C_VEL
LIN {X 0,Y 570.714,Z 278.672,A -85,B 0,C 180,E1 26244.039,E2 26244.039} C_VEL
LIN {X 0,Y 571.807,Z 280.668,A -85,B 0,C 180,E1 26243.644,E2 26243.644} C_VEL
LIN {X 0,Y 574.197,Z 285.668,A -85,B 0,C 180,E1 26242.731,E2 26242.731} C_VEL
LIN {X 0,Y 581.498,Z 295.691,A -85,B 0,C 180,E1 26241.519,E2 26241.519} C_VEL
LIN {X 0,Y 591.388,Z 309.353,A -85,B 0,C 180,E1 26240.022,E2 26240.022} C_VEL
LIN {X 0,Y 602.619,Z 325.926,A -85,B 0,C 180,E1 26238.417,E2 26238.417} C_VEL
LIN {X 0,Y 614.621,Z 345.106,A -85,B 0,C 180,E1 26236.804,E2 26236.804} C_VEL
LIN {X 0,Y 614.982,Z 346.374,A -85,B 0,C 180,E1 26236.745,E2 26236.745} C_VEL
LIN {X 0,Y 608.622,Z 578.686,A -85,B 0,C 180,E1 26233.517,E2 26233.517} C_VEL
LIN {X 0,Y 604.86,Z 720.586,A -85,B 0,C 180,E1 26231.558,E2 26231.558} C_VEL
LIN {X 0,Y 603.333,Z 747.775,A -85,B 0,C 180,E1 26231.038,E2 26231.038} C_VEL
LIN {X 0,Y 601.572,Z 771.034,A -85,B 0,C 180,E1 26230.429,E2 26230.429} C_VEL
LIN {X 0,Y 599.637,Z 792.825,A -85,B 0,C 180,E1 26229.722,E2 26229.722} C_VEL
LIN {X 0,Y 596.933,Z 819.21,A -85,B 0,C 180,E1 26228.667,E2 26228.667} C_VEL
LIN {X 0,Y 594.647,Z 838.718,A -85,B 0,C 180,E1 26227.738,E2 26227.738} C_VEL
LIN {X 0,Y 592.171,Z 858.564,A -85,B 0,C 180,E1 26226.653,E2 26226.653} C_VEL
LIN {X 0,Y 589.094,Z 881.799,A -85,B 0,C 180,E1 26225.187,E2 26225.187} C_VEL
LIN {X 0,Y 586.23,Z 901.906,A -85,B 0,C 180,E1 26223.711,E2 26223.711} C_VEL
LIN {X 0,Y 583.693,Z 919.492,A -85,B 0,C 180,E1 26222.259,E2 26222.259} C_VEL
LIN {X 0,Y 580.69,Z 940.367,A -85,B 0,C 180,E1 26220.299,E2 26220.299} C_VEL
LIN {X 0,Y 578.284,Z 957.093,A -85,B 0,C 180,E1 26218.504,E2 26218.504} C_VEL
LIN {X 0,Y 576.204,Z 972.08,A -85,B 0,C 180,E1 26216.708,E2 26216.708} C_VEL
LIN {X 0,Y 573.864,Z 989.786,A -85,B 0,C 180,E1 26214.28,E2 26214.28} C_VEL
LIN {X 0,Y 572.283,Z 1002.544,A -85,B 0,C 180,E1 26212.28,E2 26212.28} C_VEL
LIN {X 0,Y 570.886,Z 1015.594,A -85,B 0,C 180,E1 26209.97,E2 26209.97} C_VEL
LIN {X 0,Y 569.766,Z 1027.18,A -85,B 0,C 180,E1 26207.568,E2 26207.568} C_VEL
LIN {X 0,Y 569.067,Z 1035.878,A -85,B 0,C 180,E1 26205.49,E2 26205.49} C_VEL
LIN {X 0,Y 568.551,Z 1044.069,A -85,B 0,C 180,E1 26203.216,E2 26203.216} C_VEL
LIN {X 0,Y 568.183,Z 1051.877,A -85,B 0,C 180,E1 26200.546,E2 26200.546} C_VEL
LIN {X 0,Y 568.018,Z 1056.854,A -85,B 0,C 180,E1 26198.388,E2 26198.388} C_VEL
LIN {X 0,Y 567.95,Z 1060.486,A -85,B 0,C 180,E1 26196.368,E2 26196.368} C_VEL
LIN {X 0,Y 567.915,Z 1063.469,A -85,B 0,C 180,E1 26194.038,E2 26194.038} C_VEL
LIN {X 0,Y 567.901,Z 1065.19,A -85,B 0,C 180,E1 26191.412,E2 26191.412} C_VEL
LIN {X 0,Y 567.902,Z 1065.326,A -85,B 0,C 180,E1 26189.193,E2 26189.193} C_VEL
LIN {X 0,Y 567.913,Z 1064.368,A -85,B 0,C 180,E1 26187.073,E2 26187.073} C_VEL
LIN {X 0,Y 567.923,Z 1062.106,A -85,B 0,C 180,E1 26184.747,E2 26184.747} C_VEL
LIN {X 0,Y 568.004,Z 1057.861,A -85,B 0,C 180,E1 26182.108,E2 26182.108} C_VEL
LIN {X 0,Y 568.116,Z 1053.149,A -85,B 0,C 180,E1 26179.966,E2 26179.966} C_VEL
LIN {X 0,Y 568.366,Z 1047.573,A -85,B 0,C 180,E1 26177.916,E2 26177.916} C_VEL
LIN {X 0,Y 568.812,Z 1039.826,A -85,B 0,C 180,E1 26175.545,E2 26175.545} C_VEL
